//-----------------------------
//Beladestand 1
//-----------------------------
      CALL  "FC_Beladen"
      ( Stand_Nr       := 1,
        E_Belegt       := "DB_BE_Stand".Stand[1].IN_Belegt,
        E_S_innen      := "DB_BE_Stand".Stand[1].IN_innen,
        E_S_aussen     := "DB_BE_Stand".Stand[1].IN_aussen,
        E_S_verriegelt := "DB_BE_Stand".Stand[1].verriegelt,
        E_Freigabe     := "DB_BE_Stand".Stand[1].IN_Freigabe,
        Auto_Delete    := #AutoDelete,
        ext_Delete     := FALSE,
        Del_All        := #DeleteAll,
        Afg_WT_Nr      := false,
        Del_count      := 5
      );

      A     "DB_BE_Stand".Stand[1].OUT_Sperre_in;
      O     #Anforderung_QF;
      =     "DB_POS".POS[25].notFG_in;

// GO links
      L     "DB_POS".POS[27].next_WT;
      L     0;
      <>I;
      S     "DB_POS".POS[25].notFG_in;

      A     "DB_BE_Stand".Stand[1].OUT_Sperre_FW;
      O     #Sperre_TW;
      O(;
      A     "DI_FW_1".ZST.Oben_li;
      A(;
      A     "DB_BE_Stand".Stand[1].IN_Belegt;
      O     "DB_POS".POS[25].belegt;
      AN    "DB_BE_Stand".Stand[1].IN_aussen;
      );
      O;
      A     "DI_FW_1".ZST.Oben_re;
      A(;
      A     "DB_BE_Stand".Stand[2].IN_Belegt;
      O     "DB_POS".POS[26].belegt;
      AN    "DB_BE_Stand".Stand[2].IN_aussen;
      );
      );
      =     "DB_POS".POS[25].Sperre_FW;

      A     "DB_BE_Stand".Stand[1].OUT_Sperre_out;
      O     #Anforderung_QF;
      =     "DB_POS".POS[25].notFG_out;

//-----------------------------
//Beladestand 2
//-----------------------------
      CALL  "FC_Beladen"
      ( Stand_Nr       := 2,
        E_Belegt       := "DB_BE_Stand".Stand[2].IN_Belegt,
        E_S_innen      := "DB_BE_Stand".Stand[2].IN_innen,
        E_S_aussen     := "DB_BE_Stand".Stand[2].IN_aussen,
        E_S_verriegelt := "DB_BE_Stand".Stand[2].verriegelt,
        E_Freigabe     := "DB_BE_Stand".Stand[2].IN_Freigabe,
        Auto_Delete    := #AutoDelete,
        ext_Delete     := FALSE,
        Del_All        := #DeleteAll,
        Afg_WT_Nr      := false,
        Del_count      := 5
      );

      A     "DB_BE_Stand".Stand[2].OUT_Sperre_in;
      O     #Anforderung_QF;
      =     "DB_POS".POS[26].notFG_in;
// GO rechts
      L     "DB_POS".POS[28].next_WT;
      L     0;
      <>I;
      S     "DB_POS".POS[26].notFG_in;

      A     "DB_BE_Stand".Stand[2].OUT_Sperre_out;
      O     #Anforderung_QF;
      =     "DB_POS".POS[26].notFG_out;

//-----------------------------
//Beladestand 3 (GO links)
//-----------------------------
      CALL  "FC_Beladen"
      ( Stand_Nr       := 3,
        E_Belegt       := "DB_BE_Stand".Stand[3].IN_Belegt,
        E_S_innen      := "DB_BE_Stand".Stand[3].IN_innen,
        E_S_aussen     := "DB_BE_Stand".Stand[3].IN_aussen,
        E_S_verriegelt := "DB_BE_Stand".Stand[3].verriegelt,
        E_Freigabe     := "DB_BE_Stand".Stand[3].IN_Freigabe,
        Auto_Delete    := #AutoDelete,
        ext_Delete     := FALSE,
        Del_All        := #DeleteAll,
        Afg_WT_Nr      := false,
        Del_count      := 5
      );

      A     "DB_BE_Stand".Stand[3].OUT_Sperre_in;
      O     #Anforderung_QF;
      =     "DB_POS".POS[27].notFG_in;

//KS links
      L     "DB_POS".POS[25].next_WT;
      L     0;
      <>I;
      O(;
      L     "DB_POS".POS[29].next_WT;
      <>I;
      );
      O(;
      A     "DB_BE_Stand".Stand[1].IN_Belegt;
      A     "DB_BE_Stand".Stand[1].IN_innen;
      );
      O(;
      A     "DB_BE_Stand".Stand[5].IN_Belegt;
      A     "DB_BE_Stand".Stand[5].IN_innen;
      );
      S     "DB_POS".POS[27].notFG_in;

      A     "DB_BE_Stand".Stand[3].OUT_Sperre_out;
      O     #Anforderung_QF;
      =     "DB_POS".POS[27].notFG_out;

//-----------------------------
//Beladestand 4 (GO rechts)
//-----------------------------
      CALL  "FC_Beladen"
      ( Stand_Nr       := 4,
        E_Belegt       := "DB_BE_Stand".Stand[4].IN_Belegt,
        E_S_innen      := "DB_BE_Stand".Stand[4].IN_innen,
        E_S_aussen     := "DB_BE_Stand".Stand[4].IN_aussen,
        E_S_verriegelt := "DB_BE_Stand".Stand[4].verriegelt,
        E_Freigabe     := "DB_BE_Stand".Stand[4].IN_Freigabe,
        Auto_Delete    := #AutoDelete,
        ext_Delete     := FALSE,
        Del_All        := #DeleteAll,
        Afg_WT_Nr      := false,
        Del_count      := 5
      );

      A     "DB_BE_Stand".Stand[4].OUT_Sperre_in;
      O     #Anforderung_QF;
      =     "DB_POS".POS[28].notFG_in;
//KS rechts
      L     "DB_POS".POS[26].next_WT;
      L     0;
      <>I;
      O(;
      L     "DB_POS".POS[30].next_WT;
      <>I;
      );
      O(;
      A     "DB_BE_Stand".Stand[2].IN_Belegt;
      A     "DB_BE_Stand".Stand[2].IN_innen;
      );
      O(;
      A     "DB_BE_Stand".Stand[6].IN_Belegt;
      A     "DB_BE_Stand".Stand[6].IN_innen;
      );
      S     "DB_POS".POS[28].notFG_in;

      A     "DB_BE_Stand".Stand[4].OUT_Sperre_out;
      O     #Anforderung_QF;
      =     "DB_POS".POS[28].notFG_out;

//-------------------------------
//Beladestand 5 (KS hinten links)
//-------------------------------
      CALL  "FC_Beladen"
      ( Stand_Nr       := 5,
        E_Belegt       := "DB_BE_Stand".Stand[5].IN_Belegt,
        E_S_innen      := "DB_BE_Stand".Stand[5].IN_innen,
        E_S_aussen     := "DB_BE_Stand".Stand[5].IN_aussen,
        E_S_verriegelt := "DB_BE_Stand".Stand[5].verriegelt,
        E_Freigabe     := "DB_BE_Stand".Stand[5].IN_Freigabe,
        Auto_Delete    := #AutoDelete,
        ext_Delete     := FALSE,
        Del_All        := #DeleteAll,
        Afg_WT_Nr      := false,
        Del_count      := 5
      );

      L     "DB_POS".POS[25].next_WT;
      L     0;
      <>I;
      O     "DB_BE_Stand".Stand[1].IN_Belegt;
      AN    "DB_BE_Stand".Stand[1].IN_aussen;
      O     "DB_BE_Stand".Stand[5].OUT_Sperre_in;
      O     #Anforderung_QF;
      =     "DB_POS".POS[29].notFG_in;
// GO links
      L     "DB_POS".POS[27].next_WT;
      L     0;
      <>I;
      S     "DB_POS".POS[29].notFG_in;

      A     "DB_BE_Stand".Stand[5].OUT_Sperre_FW;
      O(;
      A     "DB_POS".POS[29].FW_in_POS;
      A(;
      A     "DI_FW_1".ZST.Oben_li;
      A(;
      A     "DB_BE_Stand".Stand[1].IN_Belegt;
      O     "DB_POS".POS[25].belegt;
      AN    "DB_BE_Stand".Stand[1].IN_aussen;
      );
      O;
      A     "DI_FW_1".ZST.Oben_re;
      A(;
      A     "DB_BE_Stand".Stand[2].IN_Belegt;
      O     "DB_POS".POS[26].belegt;
      AN    "DB_BE_Stand".Stand[2].IN_aussen;
      );
      );
      );
      O     #Sperre_TW;
      =     "DB_POS".POS[29].Sperre_FW;

      L     "DB_POS".POS[25].next_WT;
      L     0;
      <>I;
      O     "DB_BE_Stand".Stand[1].IN_Belegt;
      AN    "DB_BE_Stand".Stand[1].IN_aussen;
      O     "DB_BE_Stand".Stand[5].OUT_Sperre_out;
      O     #Anforderung_QF;
      =     "DB_POS".POS[29].notFG_out;

//--------------------------------
//Beladestand 6 (KS hinten rechts)
//--------------------------------
      CALL  "FC_Beladen"
      ( Stand_Nr       := 6,
        E_Belegt       := "DB_BE_Stand".Stand[6].IN_Belegt,
        E_S_innen      := "DB_BE_Stand".Stand[6].IN_innen,
        E_S_aussen     := "DB_BE_Stand".Stand[6].IN_aussen,
        E_S_verriegelt := "DB_BE_Stand".Stand[6].verriegelt,
        E_Freigabe     := "DB_BE_Stand".Stand[6].IN_Freigabe,
        Auto_Delete    := #AutoDelete,
        ext_Delete     := FALSE,
        Del_All        := #DeleteAll,
        Afg_WT_Nr      := false,
        Del_count      := 5
      );


      L     "DB_POS".POS[26].next_WT;
      L     0;
      <>I;
      O     "DB_BE_Stand".Stand[2].IN_Belegt;
      AN    "DB_BE_Stand".Stand[2].IN_aussen;
      O     "DB_BE_Stand".Stand[6].OUT_Sperre_in;
      O     #Anforderung_QF;
      =     "DB_POS".POS[30].notFG_in;
// GO rechts
      L     "DB_POS".POS[28].next_WT;
      L     0;
      <>I;
      S     "DB_POS".POS[30].notFG_in;

      L     "DB_POS".POS[26].next_WT;
      L     0;
      <>I;
      O     "DB_BE_Stand".Stand[2].IN_Belegt;
      AN    "DB_BE_Stand".Stand[2].IN_aussen;
      O     "DB_BE_Stand".Stand[6].OUT_Sperre_out;
      O     #Anforderung_QF;
      =     "DB_POS".POS[30].notFG_out;

END_FUNCTION

FUNCTION "FC_Rez_to_DB45" : Void   // FC1, LAD
TITLE = Füllt nach Aufgabetaste (Panel) Technologie DB
{ S7_Optimized_Access := 'TRUE' }
// stored: SetENOAutomatically true
   VAR_TEMP
      Ptr_Befehl_dyn : Int;
      Ptr_Param_dyn : Int;
      i : Int;
   END_VAR
   VAR CONSTANT
      KS : USInt := 1;   // kurz schmal
      LS : USInt := 2;   // lang schmal
      GO : USInt := 3;   // Großoptik
      Typ_KS : Byte := 16#11;
      Typ_LS : Byte := 16#12;
      Typ_GO : Byte := 16#20;
      Startpos_CM01 : Byte := 16#1;
      Startpos_CM02 : Byte := 16#D;
      Startpos_CM03 : Byte := 16#7;
      Startpos_CM04 : Byte := 16#13;
      Startpos_BE : Byte := 16#19;
      Laenge : Byte := 16#6;
      leer : Byte;
      M_area : Byte := 16#83;
      DB_area : Byte := 16#84;
      Ptr_Befehl_1 : Int := 260;   // Adresse Befehlsparameter
      Ptr_Befehl_2 : Int := 264;   // Adresse Befehlsparameter
      Ptr_Befehl_3 : Int := 268;   // Adresse Befehlsparameter
      Ptr_Befehl_4 : Int := 272;   // Adresse Befehlsparameter
      Ptr_Befehl_5 : Int := 276;   // Adresse Befehlsparameter
      Ptr_Befehl_6 : Int := 280;   // Adresse Befehlsparameter
      Ptr_Befehl_7 : Int;   // Adresse Befehlsparameter
      Techno_DB : DInt := 45;
   END_VAR
BEGIN

REGION Network 1 (SCL): aktuelle Auswahl in Arbeitsstruktur kopieren
   IF "DB_Prog_edit".akt_Aufgabe_Prog <> "DB_Prog_edit".old_Aufgabe_Prog THEN
       "DB_Prog_edit".Prog_Aufgabe.Prog := "DB_Prog_edit".Prog["DB_Prog_edit".akt_Aufgabe_Prog];

       "DB_Prog_edit".old_Aufgabe_Prog := "DB_Prog_edit".akt_Aufgabe_Prog;
   END_IF;
END_REGION

REGION Network 2 (SCL): Artikeldaten für aufgabe aufbereiten
   IF "Panel".Aufgabe.Freigabe AND "DB_Prog_edit".StandNr <> 0  AND "DB_Prog_edit".akt_Aufgabe_Prog <>0  AND "DB_Prog_edit".Prog_Aufgabe.Korb_Nr <>0 THEN

       "DB_Prog_edit".GZ_Charge := "DB_Prog_edit".GZ_Charge + 1; // Gesamtzähler erhöhen
       "DB_Techno".WT_NR_lng := "DB_Prog_edit".GZ_Charge; // Chargenzähler
       "DB_Techno".STAND_NR := "DB_Prog_edit".StandNr; // Nummer B/E-Stand: 1..6
       "DB_Techno".Korb_Nr := INT_TO_USINT("DB_Prog_edit".Prog_Aufgabe.Korb_Nr); // Korb 1..13

       // Modus auswerten
       IF NOT "DB_ANLAGE".config.NormalB THEN
           // Kombi-Mode
           CASE "DB_Prog_edit".Prog_Aufgabe.Korb_Nr OF
               1..3:  // "151" Korb kurz 1..3
                   "DB_Prog_edit".Prog_Aufgabe.Prog.ParaByte.%X4 := TRUE;
                   "DB_Prog_edit".Prog_Aufgabe.Prog.ParaByte.%X5 := FALSE;

               4..8:   // "161" Korb kurz 4..8
                   "DB_Prog_edit".Prog_Aufgabe.Prog.ParaByte.%X4 := FALSE;
                   "DB_Prog_edit".Prog_Aufgabe.Prog.ParaByte.%X5 := TRUE;

               9..11:  // "151" Korb lang 1..3
                   "DB_Prog_edit".Prog_Aufgabe.Prog.ParaByte.%X4 := TRUE;
                   "DB_Prog_edit".Prog_Aufgabe.Prog.ParaByte.%X5 := FALSE;

               12..13:   // "161" Korb lang 4, Großoptik 
                   "DB_Prog_edit".Prog_Aufgabe.Prog.ParaByte.%X4 := FALSE;
                   "DB_Prog_edit".Prog_Aufgabe.Prog.ParaByte.%X5 := TRUE;
           END_CASE;

       ELSE
           // Normalbetrieb
           "DB_Prog_edit".Prog_Aufgabe.Prog.ParaByte.%X4 := FALSE;
           "DB_Prog_edit".Prog_Aufgabe.Prog.ParaByte.%X5 := FALSE;
       END_IF;

       "DB_Techno".Technologie := "DB_Prog_edit".akt_Aufgabe_Prog; // aktuelles Programm: 1..99
           // WT-Typ
       CASE "DB_Prog_edit".Prog_Aufgabe.Prog.Geometrie OF
           #KS:  
               "DB_Techno".WT_Typ := #Typ_KS;
           #LS:  
               "DB_Techno".WT_Typ := #Typ_LS;
           #GO:
               "DB_Techno".WT_Typ := #Typ_GO;
           ELSE
               "DB_Techno".WT_Typ := 0;
       END_CASE;
    // Langsam senken /Langsam heben / Modi
       "DB_Techno".ParaByte := "DB_Prog_edit".Prog_Aufgabe.Prog.ParaByte;

       "DB_Techno".KorrATZ := "DB_Prog_edit".Prog_Aufgabe.Prog.Faktor_ATZ;
       "DB_Techno".KorrPend := 1.0;


       // Normal-Betrieb - nur Ware "151" Gruppe CM01/CM02
       IF "DB_ANLAGE".config.NormalB THEN
           REGION NormalB
               // Vorspülen
               #Ptr_Befehl_dyn := 1;
               #Ptr_Param_dyn := 340;

               "DB_Techno".stBefehle[#Ptr_Befehl_dyn].Kennung := #Startpos_CM03;
               "DB_Techno".stBefehle[#Ptr_Befehl_dyn].FirstPos1 := #Startpos_CM03;
               "DB_Techno".stBefehle[#Ptr_Befehl_dyn].Grpleng1 := #Laenge;
               "DB_Techno".stBefehle[#Ptr_Befehl_dyn].FirstPos2 := #leer;
               "DB_Techno".stBefehle[#Ptr_Befehl_dyn].Grpleng2 := #leer;
               "DB_Techno".stBefehle[#Ptr_Befehl_dyn].Merker := #leer;
               "DB_Techno".stBefehle[#Ptr_Befehl_dyn].Param_Ptr := #Ptr_Param_dyn; //#Ptr_Befehl_1;
               "temp_Sollzeit" := TOD_TO_DINT("DB_Prog_edit".Prog_Aufgabe.Prog.CM03_VorSpuel.Expo) / 1000;

               POKE_BLK(area_src := #M_area,
                        dbNumber_src := 0,
                        byteOffset_src := 256,
                        area_dest := #DB_area,
                        dbNumber_dest := #Techno_DB,
                        byteOffset_dest := #Ptr_Param_dyn, //Ptr_Befehl_1,
                        count := 4);

               // Vorätzen
               IF "DB_Prog_edit".Prog_Aufgabe.Prog.CM01_VorAetz.Anzahl_Voraetz > 0 THEN
                   FOR #i := 1 TO BYTE_TO_INT("DB_Prog_edit".Prog_Aufgabe.Prog.CM01_VorAetz.Anzahl_Voraetz) DO
                       #Ptr_Befehl_dyn := #Ptr_Befehl_dyn + 1;
                       #Ptr_Param_dyn := #Ptr_Param_dyn + 4;

                       "DB_Techno".stBefehle[#Ptr_Befehl_dyn].Kennung := #Startpos_CM01;
                       "DB_Techno".stBefehle[#Ptr_Befehl_dyn].FirstPos1 := #Startpos_CM01;
                       "DB_Techno".stBefehle[#Ptr_Befehl_dyn].Grpleng1 := #Laenge;
                       "DB_Techno".stBefehle[#Ptr_Befehl_dyn].FirstPos2 := #Startpos_CM02;
                       "DB_Techno".stBefehle[#Ptr_Befehl_dyn].Grpleng2 := #Laenge;
                       "DB_Techno".stBefehle[#Ptr_Befehl_dyn].Merker := #leer;
                       "DB_Techno".stBefehle[#Ptr_Befehl_dyn].Param_Ptr := #Ptr_Param_dyn; // #Ptr_Befehl_2;
                       "temp_Sollzeit" := TOD_TO_DINT("DB_Prog_edit".Prog_Aufgabe.Prog.CM01_VorAetz.Expo) / 1000;

                       POKE_BLK(area_src := #M_area,
                                dbNumber_src := 0,
                                byteOffset_src := 256,
                                area_dest := #DB_area,
                                dbNumber_dest := #Techno_DB,
                                byteOffset_dest := #Ptr_Param_dyn, //Ptr_Befehl_2,
                                count := 4);


                       // Spülen Vorätzen
                       #Ptr_Befehl_dyn := #Ptr_Befehl_dyn + 1;
                       #Ptr_Param_dyn := #Ptr_Param_dyn + 4;

                       "DB_Techno".stBefehle[#Ptr_Befehl_dyn].Kennung := #Startpos_CM03;
                       "DB_Techno".stBefehle[#Ptr_Befehl_dyn].FirstPos1 := #Startpos_CM03;
                       "DB_Techno".stBefehle[#Ptr_Befehl_dyn].Grpleng1 := #Laenge;
                       "DB_Techno".stBefehle[#Ptr_Befehl_dyn].FirstPos2 := #leer;
                       "DB_Techno".stBefehle[#Ptr_Befehl_dyn].Grpleng2 := #leer;
                       "DB_Techno".stBefehle[#Ptr_Befehl_dyn].Merker := #leer;
                       "DB_Techno".stBefehle[#Ptr_Befehl_dyn].Param_Ptr := #Ptr_Param_dyn; // #Ptr_Befehl_3;
                       "temp_Sollzeit" := TOD_TO_DINT("DB_Prog_edit".Prog_Aufgabe.Prog.CM03_SpuelVorAetz.Expo) / 1000;

                       POKE_BLK(area_src := #M_area,
                                dbNumber_src := 0,
                                byteOffset_src := 256,
                                area_dest := #DB_area,
                                dbNumber_dest := #Techno_DB,
                                byteOffset_dest := #Ptr_Param_dyn, //#Ptr_Befehl_3,
                                count := 4);

                   END_FOR;
               END_IF;

               // Ätzen
               #Ptr_Befehl_dyn := #Ptr_Befehl_dyn + 1;
               #Ptr_Param_dyn := #Ptr_Param_dyn + 4;

               "DB_Techno".stBefehle[#Ptr_Befehl_dyn].Kennung := #Startpos_CM01;
               "DB_Techno".stBefehle[#Ptr_Befehl_dyn].FirstPos1 := #Startpos_CM01;
               "DB_Techno".stBefehle[#Ptr_Befehl_dyn].Grpleng1 := #Laenge;
               "DB_Techno".stBefehle[#Ptr_Befehl_dyn].FirstPos2 := #Startpos_CM02;
               "DB_Techno".stBefehle[#Ptr_Befehl_dyn].Grpleng2 := #Laenge;
               "DB_Techno".stBefehle[#Ptr_Befehl_dyn].Merker := #leer;
               "DB_Techno".stBefehle[#Ptr_Befehl_dyn].Param_Ptr := #Ptr_Param_dyn; //#Ptr_Befehl_4;
               "temp_Sollzeit" := TOD_TO_DINT("DB_Prog_edit".Prog_Aufgabe.Prog.CM01_Aetzen.Expo) / 1000;

               POKE_BLK(area_src := #M_area,
                        dbNumber_src := 0,
                        byteOffset_src := 256,
                        area_dest := #DB_area,
                        dbNumber_dest := #Techno_DB,
                        byteOffset_dest := #Ptr_Param_dyn, //#Ptr_Befehl_4,
                        count := 4);

               // Spülen 1 Ätzen
               #Ptr_Befehl_dyn := #Ptr_Befehl_dyn + 1;
               #Ptr_Param_dyn := #Ptr_Param_dyn + 4;

               "DB_Techno".stBefehle[#Ptr_Befehl_dyn].Kennung := #Startpos_CM03;
               "DB_Techno".stBefehle[#Ptr_Befehl_dyn].FirstPos1 := #Startpos_CM03;
               "DB_Techno".stBefehle[#Ptr_Befehl_dyn].Grpleng1 := #Laenge;
               "DB_Techno".stBefehle[#Ptr_Befehl_dyn].FirstPos2 := #leer;
               "DB_Techno".stBefehle[#Ptr_Befehl_dyn].Grpleng2 := #leer;
               "DB_Techno".stBefehle[#Ptr_Befehl_dyn].Merker := #leer;
               "DB_Techno".stBefehle[#Ptr_Befehl_dyn].Param_Ptr := #Ptr_Param_dyn; //#Ptr_Befehl_5;
               "temp_Sollzeit" := TOD_TO_DINT("DB_Prog_edit".Prog_Aufgabe.Prog.CM03_Spl_1.Expo) / 1000;

               POKE_BLK(area_src := #M_area,
                        dbNumber_src := 0,
                        byteOffset_src := 256,
                        area_dest := #DB_area,
                        dbNumber_dest := #Techno_DB,
                        byteOffset_dest := #Ptr_Param_dyn, //#Ptr_Befehl_5,
                        count := 4);

               // Spülen 2 Ätzen
               #Ptr_Befehl_dyn := #Ptr_Befehl_dyn + 1;
               #Ptr_Param_dyn := #Ptr_Param_dyn + 4;

               "DB_Techno".stBefehle[#Ptr_Befehl_dyn].Kennung := #Startpos_CM04;
               "DB_Techno".stBefehle[#Ptr_Befehl_dyn].FirstPos1 := #Startpos_CM04;
               "DB_Techno".stBefehle[#Ptr_Befehl_dyn].Grpleng1 := #Laenge;
               "DB_Techno".stBefehle[#Ptr_Befehl_dyn].FirstPos2 := #leer;
               "DB_Techno".stBefehle[#Ptr_Befehl_dyn].Grpleng2 := #leer;
               "DB_Techno".stBefehle[#Ptr_Befehl_dyn].Merker := #leer;
               "DB_Techno".stBefehle[#Ptr_Befehl_dyn].Param_Ptr := #Ptr_Param_dyn; //#Ptr_Befehl_6;
               "temp_Sollzeit" := TOD_TO_DINT("DB_Prog_edit".Prog_Aufgabe.Prog.CM04_Spl_2.Expo) / 1000;

               POKE_BLK(area_src := #M_area,
                        dbNumber_src := 0,
                        byteOffset_src := 256,
                        area_dest := #DB_area,
                        dbNumber_dest := #Techno_DB,
                        byteOffset_dest := #Ptr_Param_dyn, //#Ptr_Befehl_6,
                        count := 4);
           END_REGION

       ELSE // Kombi-Modus: "151" CM02 / CM04 ; "161" CM01 / CM03


           IF  "DB_Prog_edit".Prog_Aufgabe.Prog.ParaByte.%X4 THEN
            REGION WT_151                    
                // Vorspülen             
                  #Ptr_Befehl_dyn := 1;
                  #Ptr_Param_dyn := 340;

                  "DB_Techno".stBefehle[#Ptr_Befehl_dyn].Kennung := #Startpos_CM04;
                   "DB_Techno".stBefehle[#Ptr_Befehl_dyn].FirstPos1 := #Startpos_CM04;
                   "DB_Techno".stBefehle[#Ptr_Befehl_dyn].Grpleng1 := #Laenge;
                   "DB_Techno".stBefehle[#Ptr_Befehl_dyn].FirstPos2 := #leer;
                   "DB_Techno".stBefehle[#Ptr_Befehl_dyn].Grpleng2 := #leer;
                   "DB_Techno".stBefehle[#Ptr_Befehl_dyn].Merker := #leer;
                   "DB_Techno".stBefehle[#Ptr_Befehl_dyn].Param_Ptr := #Ptr_Param_dyn; //#Ptr_Befehl_1;
                   "temp_Sollzeit" := TOD_TO_DINT("DB_Prog_edit".Prog_Aufgabe.Prog.CM03_VorSpuel.Expo) / 1000;

                   POKE_BLK(area_src := #M_area,
                            dbNumber_src := 0,
                            byteOffset_src := 256,
                            area_dest := #DB_area,
                            dbNumber_dest := #Techno_DB,
                            byteOffset_dest := #Ptr_Param_dyn, //Ptr_Befehl_1,
                            count := 4);

                   // Vorätzen
                   IF "DB_Prog_edit".Prog_Aufgabe.Prog.CM01_VorAetz.Anzahl_Voraetz > 0 THEN
                       FOR #i := 1 TO BYTE_TO_INT("DB_Prog_edit".Prog_Aufgabe.Prog.CM01_VorAetz.Anzahl_Voraetz) DO
                           #Ptr_Befehl_dyn := #Ptr_Befehl_dyn + 1;
                           #Ptr_Param_dyn := #Ptr_Param_dyn + 4;

                           "DB_Techno".stBefehle[#Ptr_Befehl_dyn].Kennung := #Startpos_CM02;
                           "DB_Techno".stBefehle[#Ptr_Befehl_dyn].FirstPos1 := #Startpos_CM02;
                           "DB_Techno".stBefehle[#Ptr_Befehl_dyn].Grpleng1 := #Laenge;
                           "DB_Techno".stBefehle[#Ptr_Befehl_dyn].FirstPos2 := #leer;
                           "DB_Techno".stBefehle[#Ptr_Befehl_dyn].Grpleng2 := #leer;
                           "DB_Techno".stBefehle[#Ptr_Befehl_dyn].Merker := #leer;
                           "DB_Techno".stBefehle[#Ptr_Befehl_dyn].Param_Ptr := #Ptr_Param_dyn; // #Ptr_Befehl_2;
                           "temp_Sollzeit" := TOD_TO_DINT("DB_Prog_edit".Prog_Aufgabe.Prog.CM01_VorAetz.Expo) / 1000;

                           POKE_BLK(area_src := #M_area,
                                    dbNumber_src := 0,
                                    byteOffset_src := 256,
                                    area_dest := #DB_area,
                                    dbNumber_dest := #Techno_DB,
                                    byteOffset_dest := #Ptr_Param_dyn, //Ptr_Befehl_2,
                                    count := 4);

                           // Spülen Vorätzen
                           #Ptr_Befehl_dyn := #Ptr_Befehl_dyn + 1;
                           #Ptr_Param_dyn := #Ptr_Param_dyn + 4;

                           "DB_Techno".stBefehle[#Ptr_Befehl_dyn].Kennung := #Startpos_CM04;
                           "DB_Techno".stBefehle[#Ptr_Befehl_dyn].FirstPos1 := #Startpos_CM04;
                           "DB_Techno".stBefehle[#Ptr_Befehl_dyn].Grpleng1 := #Laenge;
                           "DB_Techno".stBefehle[#Ptr_Befehl_dyn].FirstPos2 := #leer;
                           "DB_Techno".stBefehle[#Ptr_Befehl_dyn].Grpleng2 := #leer;
                           "DB_Techno".stBefehle[#Ptr_Befehl_dyn].Merker := #leer;
                           "DB_Techno".stBefehle[#Ptr_Befehl_dyn].Param_Ptr := #Ptr_Param_dyn; // #Ptr_Befehl_3;
                           "temp_Sollzeit" := TOD_TO_DINT("DB_Prog_edit".Prog_Aufgabe.Prog.CM03_SpuelVorAetz.Expo) / 1000;

                           POKE_BLK(area_src := #M_area,
                                    dbNumber_src := 0,
                                    byteOffset_src := 256,
                                    area_dest := #DB_area,
                                    dbNumber_dest := #Techno_DB,
                                    byteOffset_dest := #Ptr_Param_dyn, //#Ptr_Befehl_3,
                                    count := 4);

                       END_FOR;
                   END_IF;

                   // Ätzen
                   #Ptr_Befehl_dyn := #Ptr_Befehl_dyn + 1;
                   #Ptr_Param_dyn := #Ptr_Param_dyn + 4;

                   "DB_Techno".stBefehle[#Ptr_Befehl_dyn].Kennung := #Startpos_CM02;
                   "DB_Techno".stBefehle[#Ptr_Befehl_dyn].FirstPos1 := #Startpos_CM02;
                   "DB_Techno".stBefehle[#Ptr_Befehl_dyn].Grpleng1 := #Laenge;
                   "DB_Techno".stBefehle[#Ptr_Befehl_dyn].FirstPos2 := #leer;
                   "DB_Techno".stBefehle[#Ptr_Befehl_dyn].Grpleng2 := #leer;
                   "DB_Techno".stBefehle[#Ptr_Befehl_dyn].Merker := #leer;
                   "DB_Techno".stBefehle[#Ptr_Befehl_dyn].Param_Ptr := #Ptr_Param_dyn; //#Ptr_Befehl_4;
                   "temp_Sollzeit" := TOD_TO_DINT("DB_Prog_edit".Prog_Aufgabe.Prog.CM01_Aetzen.Expo) / 1000;

                   POKE_BLK(area_src := #M_area,
                            dbNumber_src := 0,
                            byteOffset_src := 256,
                            area_dest := #DB_area,
                            dbNumber_dest := #Techno_DB,
                            byteOffset_dest := #Ptr_Param_dyn, //#Ptr_Befehl_4,
                            count := 4);

                   // Spülen 1 Ätzen
                   #Ptr_Befehl_dyn := #Ptr_Befehl_dyn + 1;
                   #Ptr_Param_dyn := #Ptr_Param_dyn + 4;

                   "DB_Techno".stBefehle[#Ptr_Befehl_dyn].Kennung := #Startpos_CM04;
                   "DB_Techno".stBefehle[#Ptr_Befehl_dyn].FirstPos1 := #Startpos_CM04;
                   "DB_Techno".stBefehle[#Ptr_Befehl_dyn].Grpleng1 := #Laenge;
                   "DB_Techno".stBefehle[#Ptr_Befehl_dyn].FirstPos2 := #leer;
                   "DB_Techno".stBefehle[#Ptr_Befehl_dyn].Grpleng2 := #leer;
                   "DB_Techno".stBefehle[#Ptr_Befehl_dyn].Merker := #leer;
                   "DB_Techno".stBefehle[#Ptr_Befehl_dyn].Param_Ptr := #Ptr_Param_dyn; //#Ptr_Befehl_5;
                   "temp_Sollzeit" := TOD_TO_DINT("DB_Prog_edit".Prog_Aufgabe.Prog.CM03_Spl_1.Expo) / 1000;

                   POKE_BLK(area_src := #M_area,
                            dbNumber_src := 0,
                            byteOffset_src := 256,
                            area_dest := #DB_area,
                            dbNumber_dest := #Techno_DB,
                            byteOffset_dest := #Ptr_Param_dyn, //#Ptr_Befehl_5,
                            count := 4);

                   // Spülen 2 Ätzen
                   #Ptr_Befehl_dyn := #Ptr_Befehl_dyn + 1;
                   #Ptr_Param_dyn := #Ptr_Param_dyn + 4;

                   "DB_Techno".stBefehle[#Ptr_Befehl_dyn].Kennung := #Startpos_CM04;
                   "DB_Techno".stBefehle[#Ptr_Befehl_dyn].FirstPos1 := #Startpos_CM04;
                   "DB_Techno".stBefehle[#Ptr_Befehl_dyn].Grpleng1 := #Laenge;
                   "DB_Techno".stBefehle[#Ptr_Befehl_dyn].FirstPos2 := #leer;
                   "DB_Techno".stBefehle[#Ptr_Befehl_dyn].Grpleng2 := #leer;
                   "DB_Techno".stBefehle[#Ptr_Befehl_dyn].Merker := #leer;
                   "DB_Techno".stBefehle[#Ptr_Befehl_dyn].Param_Ptr := #Ptr_Param_dyn; //#Ptr_Befehl_6;
                   "temp_Sollzeit" := TOD_TO_DINT("DB_Prog_edit".Prog_Aufgabe.Prog.CM04_Spl_2.Expo) / 1000;

                   POKE_BLK(area_src := #M_area,
                            dbNumber_src := 0,
                            byteOffset_src := 256,
                            area_dest := #DB_area,
                            dbNumber_dest := #Techno_DB,
                            byteOffset_dest := #Ptr_Param_dyn, //#Ptr_Befehl_6,
                            count := 4);
               END_REGION

           ELSE
            REGION WT_161                    
                   // Vorspülen             
                   #Ptr_Befehl_dyn := 1;
                   #Ptr_Param_dyn := 340;

                   "DB_Techno".stBefehle[#Ptr_Befehl_dyn].Kennung := #Startpos_CM03;
                   "DB_Techno".stBefehle[#Ptr_Befehl_dyn].FirstPos1 := #Startpos_CM03;
                   "DB_Techno".stBefehle[#Ptr_Befehl_dyn].Grpleng1 := #Laenge;
                   "DB_Techno".stBefehle[#Ptr_Befehl_dyn].FirstPos2 := #leer;
                   "DB_Techno".stBefehle[#Ptr_Befehl_dyn].Grpleng2 := #leer;
                   "DB_Techno".stBefehle[#Ptr_Befehl_dyn].Merker := #leer;
                   "DB_Techno".stBefehle[#Ptr_Befehl_dyn].Param_Ptr := #Ptr_Param_dyn; //#Ptr_Befehl_1;
                   "temp_Sollzeit" := TOD_TO_DINT("DB_Prog_edit".Prog_Aufgabe.Prog.CM03_VorSpuel.Expo) / 1000;

                   POKE_BLK(area_src := #M_area,
                            dbNumber_src := 0,
                            byteOffset_src := 256,
                            area_dest := #DB_area,
                            dbNumber_dest := #Techno_DB,
                            byteOffset_dest := #Ptr_Param_dyn, //Ptr_Befehl_1,
                            count := 4);

                   // Vorätzen
                   IF "DB_Prog_edit".Prog_Aufgabe.Prog.CM01_VorAetz.Anzahl_Voraetz > 0 THEN
                       FOR #i := 1 TO BYTE_TO_INT("DB_Prog_edit".Prog_Aufgabe.Prog.CM01_VorAetz.Anzahl_Voraetz) DO
                           #Ptr_Befehl_dyn := #Ptr_Befehl_dyn + 1;
                           #Ptr_Param_dyn := #Ptr_Param_dyn + 4;

                           "DB_Techno".stBefehle[#Ptr_Befehl_dyn].Kennung := #Startpos_CM01;
                           "DB_Techno".stBefehle[#Ptr_Befehl_dyn].FirstPos1 := #Startpos_CM01;
                           "DB_Techno".stBefehle[#Ptr_Befehl_dyn].Grpleng1 := #Laenge;
                           "DB_Techno".stBefehle[#Ptr_Befehl_dyn].FirstPos2 := #leer;
                           "DB_Techno".stBefehle[#Ptr_Befehl_dyn].Grpleng2 := #leer;
                           "DB_Techno".stBefehle[#Ptr_Befehl_dyn].Merker := #leer;
                           "DB_Techno".stBefehle[#Ptr_Befehl_dyn].Param_Ptr := #Ptr_Param_dyn; // #Ptr_Befehl_2;
                           "temp_Sollzeit" := TOD_TO_DINT("DB_Prog_edit".Prog_Aufgabe.Prog.CM01_VorAetz.Expo) / 1000;

                           POKE_BLK(area_src := #M_area,
                                    dbNumber_src := 0,
                                    byteOffset_src := 256,
                                    area_dest := #DB_area,
                                    dbNumber_dest := #Techno_DB,
                                    byteOffset_dest := #Ptr_Param_dyn, //Ptr_Befehl_2,
                                    count := 4);

                           // Spülen Vorätzen
                           #Ptr_Befehl_dyn := #Ptr_Befehl_dyn + 1;
                           #Ptr_Param_dyn := #Ptr_Param_dyn + 4;

                           "DB_Techno".stBefehle[#Ptr_Befehl_dyn].Kennung := #Startpos_CM03;
                           "DB_Techno".stBefehle[#Ptr_Befehl_dyn].FirstPos1 := #Startpos_CM03;
                           "DB_Techno".stBefehle[#Ptr_Befehl_dyn].Grpleng1 := #Laenge;
                           "DB_Techno".stBefehle[#Ptr_Befehl_dyn].FirstPos2 := #leer;
                           "DB_Techno".stBefehle[#Ptr_Befehl_dyn].Grpleng2 := #leer;
                           "DB_Techno".stBefehle[#Ptr_Befehl_dyn].Merker := #leer;
                           "DB_Techno".stBefehle[#Ptr_Befehl_dyn].Param_Ptr := #Ptr_Param_dyn; // #Ptr_Befehl_3;
                           "temp_Sollzeit" := TOD_TO_DINT("DB_Prog_edit".Prog_Aufgabe.Prog.CM03_SpuelVorAetz.Expo) / 1000;

                           POKE_BLK(area_src := #M_area,
                                    dbNumber_src := 0,
                                    byteOffset_src := 256,
                                    area_dest := #DB_area,
                                    dbNumber_dest := #Techno_DB,
                                    byteOffset_dest := #Ptr_Param_dyn, //#Ptr_Befehl_3,
                                    count := 4);

                       END_FOR;
                   END_IF;

                   // Ätzen
                   #Ptr_Befehl_dyn := #Ptr_Befehl_dyn + 1;
                   #Ptr_Param_dyn := #Ptr_Param_dyn + 4;

                   "DB_Techno".stBefehle[#Ptr_Befehl_dyn].Kennung := #Startpos_CM01;
                   "DB_Techno".stBefehle[#Ptr_Befehl_dyn].FirstPos1 := #Startpos_CM01;
                   "DB_Techno".stBefehle[#Ptr_Befehl_dyn].Grpleng1 := #Laenge;
                   "DB_Techno".stBefehle[#Ptr_Befehl_dyn].FirstPos2 := #leer;
                   "DB_Techno".stBefehle[#Ptr_Befehl_dyn].Grpleng2 := #leer;
                   "DB_Techno".stBefehle[#Ptr_Befehl_dyn].Merker := #leer;
                   "DB_Techno".stBefehle[#Ptr_Befehl_dyn].Param_Ptr := #Ptr_Param_dyn; //#Ptr_Befehl_4;
                   "temp_Sollzeit" := TOD_TO_DINT("DB_Prog_edit".Prog_Aufgabe.Prog.CM01_Aetzen.Expo) / 1000;

                   POKE_BLK(area_src := #M_area,
                            dbNumber_src := 0,
                            byteOffset_src := 256,
                            area_dest := #DB_area,
                            dbNumber_dest := #Techno_DB,
                            byteOffset_dest := #Ptr_Param_dyn, //#Ptr_Befehl_4,
                            count := 4);

                   // Spülen 1 Ätzen
                   #Ptr_Befehl_dyn := #Ptr_Befehl_dyn + 1;
                   #Ptr_Param_dyn := #Ptr_Param_dyn + 4;

                   "DB_Techno".stBefehle[#Ptr_Befehl_dyn].Kennung := #Startpos_CM03;
                   "DB_Techno".stBefehle[#Ptr_Befehl_dyn].FirstPos1 := #Startpos_CM03;
                   "DB_Techno".stBefehle[#Ptr_Befehl_dyn].Grpleng1 := #Laenge;
                   "DB_Techno".stBefehle[#Ptr_Befehl_dyn].FirstPos2 := #leer;
                   "DB_Techno".stBefehle[#Ptr_Befehl_dyn].Grpleng2 := #leer;
                   "DB_Techno".stBefehle[#Ptr_Befehl_dyn].Merker := #leer;
                   "DB_Techno".stBefehle[#Ptr_Befehl_dyn].Param_Ptr := #Ptr_Param_dyn; //#Ptr_Befehl_5;
                   "temp_Sollzeit" := TOD_TO_DINT("DB_Prog_edit".Prog_Aufgabe.Prog.CM03_Spl_1.Expo) / 1000;

                   POKE_BLK(area_src := #M_area,
                            dbNumber_src := 0,
                            byteOffset_src := 256,
                            area_dest := #DB_area,
                            dbNumber_dest := #Techno_DB,
                            byteOffset_dest := #Ptr_Param_dyn, //#Ptr_Befehl_5,
                            count := 4);

                   // Spülen 2 Ätzen
                   #Ptr_Befehl_dyn := #Ptr_Befehl_dyn + 1;
                   #Ptr_Param_dyn := #Ptr_Param_dyn + 4;

                   "DB_Techno".stBefehle[#Ptr_Befehl_dyn].Kennung := #Startpos_CM03;
                   "DB_Techno".stBefehle[#Ptr_Befehl_dyn].FirstPos1 := #Startpos_CM03;
                   "DB_Techno".stBefehle[#Ptr_Befehl_dyn].Grpleng1 := #Laenge;
                   "DB_Techno".stBefehle[#Ptr_Befehl_dyn].FirstPos2 := #leer;
                   "DB_Techno".stBefehle[#Ptr_Befehl_dyn].Grpleng2 := #leer;
                   "DB_Techno".stBefehle[#Ptr_Befehl_dyn].Merker := #leer;
                   "DB_Techno".stBefehle[#Ptr_Befehl_dyn].Param_Ptr := #Ptr_Param_dyn; //#Ptr_Befehl_6;
                   "temp_Sollzeit" := TOD_TO_DINT("DB_Prog_edit".Prog_Aufgabe.Prog.CM04_Spl_2.Expo) / 1000;

                   POKE_BLK(area_src := #M_area,
                            dbNumber_src := 0,
                            byteOffset_src := 256,
                            area_dest := #DB_area,
                            dbNumber_dest := #Techno_DB,
                            byteOffset_dest := #Ptr_Param_dyn, //#Ptr_Befehl_6,
                            count := 4);
               END_REGION

            END_IF;

       END_IF;

       // Ausfahrt
       #Ptr_Befehl_dyn := #Ptr_Befehl_dyn + 1;
       #Ptr_Param_dyn := #Ptr_Param_dyn + 4;

       "DB_Techno".stBefehle[#Ptr_Befehl_dyn].Kennung := #Startpos_BE;
       "DB_Techno".stBefehle[#Ptr_Befehl_dyn].FirstPos1 := #Startpos_BE;
       "DB_Techno".stBefehle[#Ptr_Befehl_dyn].Grpleng1 := #Laenge;
       "DB_Techno".stBefehle[#Ptr_Befehl_dyn].FirstPos2 := #leer;
       "DB_Techno".stBefehle[#Ptr_Befehl_dyn].Grpleng2 := #leer;
       "DB_Techno".stBefehle[#Ptr_Befehl_dyn].Merker := #leer;
       "DB_Techno".stBefehle[#Ptr_Befehl_dyn].Param_Ptr := #Ptr_Param_dyn; //#Ptr_Befehl_7;

       // Ende
       #Ptr_Befehl_dyn := #Ptr_Befehl_dyn + 1;

       FOR #i := #Ptr_Befehl_dyn TO 20 DO
            #Ptr_Befehl_dyn := #i;
            // #Ptr_Param_dyn := #Ptr_Param_dyn + 4;

           "DB_Techno".stBefehle[#Ptr_Befehl_dyn].Kennung := #leer;
           "DB_Techno".stBefehle[#Ptr_Befehl_dyn].FirstPos1 := #leer;
           "DB_Techno".stBefehle[#Ptr_Befehl_dyn].Grpleng1 := #leer;
           "DB_Techno".stBefehle[#Ptr_Befehl_dyn].FirstPos2 := #leer;
           "DB_Techno".stBefehle[#Ptr_Befehl_dyn].Grpleng2 := #leer;
           "DB_Techno".stBefehle[#Ptr_Befehl_dyn].Merker := #leer;
           "DB_Techno".stBefehle[#Ptr_Befehl_dyn].Param_Ptr := 0;
       END_FOR;

       "DB_Techno".Name := "DB_Prog_edit".Prog_Aufgabe.Prog.Name;

       "DB_Techno".DATEN_gueltig := "Panel".Aufgabe.Freigabe;
       // Rücksetzen
       "Panel".Aufgabe.Freigabe := FALSE;
       "DB_Prog_edit".StandNr := 0;
       "DB_Prog_edit".Variante := 0;
       "DB_Prog_edit".Prog_Aufgabe.Korb_Nr := 0;

   END_IF;
END_REGION
END_FUNCTION

FUNCTION "FC_AEND_WT" : Void   // FC45, STL
TITLE = WT-Daten neu/geändert
{ S7_Optimized_Access := 'FALSE' }
AUTHOR : MS
// Laden von WT-Daten aus Übergabepuffer
// stored: AutoNumber false
   VAR_TEMP
      WT_lang : DWord;
      WT_Nr_lang : DWord;
      WT_DB : Int;
      Quell_DB : Int;
      last_WT_DB : Int;
      Beginn_Daten : Int;
      Ende_daten : Int;
      Stand_Nr : USInt;
      Pos_Nr : USInt;
      WT_Nr : Byte;
      WT_kurz : Byte;
      inf_1 : Byte;
      WTnew : Bool;   // Warenträger neu
      "Return" : Bool;
      Stand_ok : Bool;
      WT_nok : Bool;
      neuAufgabe : Bool;
      Del_All : Bool;
   END_VAR
BEGIN

NETWORK
TITLE = Test gibt es neue Daten
// -gibt es neue Daten
// -wo stehen diese
// -handelt es sich um Aktualisierungsdaten
//-------------------------------
//Neue Daten?
//-------------------------------
      A     "DB_Techno".DATEN_gueltig;
      L     S5T#20S;
      SD    "T_Aend_WT";

      A     "DB_Techno".DATEN_gueltig;
      A     "T_Aend_WT";
      R     "DB_Techno".DATEN_gueltig;
//-------------------------------
//keine neuen Daten
//-------------------------------
      AN    "DB_Techno".DATEN_gueltig;
      BEC;
      SET;
      R     #Stand_ok;
      R     #Del_All;

//----------------------------------
//Handelt es sich um eine Neuaufgabe
//----------------------------------
      L     "DB_Techno".STAND_NR;
      T     #Stand_Nr;
      L     0;
      <>I;
      =     #WTnew;
      =     #neuAufgabe;
      JC    New;
      JU    Old;


NETWORK
TITLE = Neuer WT
//------------------------
//Stand-Nr prüfen
//------------------------
New:  L     "DB_BE_Stand".Anzahl;
      L     #Stand_Nr;
      <I;
      JC    ende;

      OPN   "DB_BE_Stand";
      A     "DB_BE_Stand".Stand[#Stand_Nr].Del_All;
      =     #Del_All;
      L     0;
      L     "DB_BE_Stand".Stand[#Stand_Nr].Pos_Nr;
      ==I;
      JC    ende;
      S     #Stand_ok;
//------------------------
//Pos auf WT testen
//------------------------
      T     #Pos_Nr;
      L     0;
      L     "DB_POS".POS[#Pos_Nr].WT_DB;
      ==I;
      JC    WTck;
      T     #WT_Nr;
      L     100;
      +I;
      T     #WT_DB;
      JU    load;
//------------------------
//Neuen WT suchen
//------------------------
WTck: AN    #Del_All;  //keinen neuen WT suchen
      JC    ende;
      L     "DB_ANLAGE".config.ANZ_WT;
      L     100;
      +I;
      T     #last_WT_DB;
      L     101;
      T     #WT_DB;
ret:  OPN   DB [#WT_DB];
      L     %DBB15;
      L     0;
      ==I;
      JC    fnd;
      L     #WT_DB;
      L     1;
      +I;
      T     #WT_DB;
      L     #last_WT_DB;
      >I;
      JC    ende;
      JU    ret;
fnd:  L     #WT_DB;
      L     100;
      -I;
      T     #WT_Nr;
      JU    load;


NETWORK
TITLE = Alter WT
// Aktualisieren
//-------------------------------
//prüfen ob WT_Nr gültig
//-------------------------------
Old:  L     "DB_Techno".WT_NR_kurz;
      T     #WT_Nr;
      L     "DB_ANLAGE".config.ANZ_WT;
      >I;
      JC    ende;
      L     0;
      L     #WT_Nr;
      >=I;
      JC    ende;
      L     100;
      +I;
      T     #WT_DB;
//-------------------------------
//passen die WT-Daten zueinander
//-------------------------------
      L     "DB_Techno".WT_NR_lng;
      OPN   DB [#WT_DB];
      L     %DBD6;  // WT-Nr lang
      <>D;
      JC    ende;
      L     %DBB15;  //"DB_WTx".POS
      T     #Pos_Nr;

load: NOP   0;

NETWORK
TITLE = Daten laden
//------------------------
//allgemeine Daten laden
//------------------------
ldok: L     "DB_Techno".Beginn_Daten;
      T     #Beginn_Daten;
      L     "DB_Techno".Ende_Daten;
      T     #Ende_daten;

      CALL  "FC_DB_COPY"
      ( CLR_ALT_DB := FALSE,
        ALT_DB     := 45,
        NEU_DB     := #WT_DB,
        COPY_START := #Beginn_Daten,
        COPY_ENDE  := #Ende_daten,
        ZIEL_START := 78,  // HCA: Namen mit kopieren
        CLR_START  := 0,
        CLR_ENDE   := 0,
        START      := "DB_Techno".DATEN_gueltig
      );

      L     "DB_Techno".Prioritaet;
      L     0;
      <>I;
      OPN   DB [#WT_DB];
      =     %DBX18.0;  //PRIORITÄT

      OPN   DB [#WT_DB];
      A     %DBX18.1;  //"DB_WT1".in_Anlage
      R     #neuAufgabe;  //WT wurde bereits neu aufgegeben

      A     %DBX22.3;  //"DB_WT1".WT_nok
      AN    #Stand_ok;
      =     #WT_nok;  //nok merken

      L     "DB_Techno".ParaByte;  //Parameterinfo laden
      OPN   DB [#WT_DB];
      T     %DBB22;
      L     "DB_Techno".WT_NR_lng;
      OPN   DB [#WT_DB];
      T     %DBD6;  //WT_Nr_lang
      T     #WT_Nr_lang;
      L     "DB_Techno".Speed_Up;
      OPN   DB [#WT_DB];
      T     %DBW64;  //"DB_WT1".Speed_Up
      L     "DB_Techno".Speed_Dn;
      OPN   DB [#WT_DB];
      T     %DBW66;  //"DB_WT1".Speed_Dn
      L     "DB_Techno".Speed_Fahrt;
      OPN   DB [#WT_DB];
      T     %DBW68;  //"DB_WT1".Speed_Fahrt
      L     "DB_Techno".KorrPend;  //Korrektur Pendeln laden
      OPN   DB [#WT_DB];
      T     %DBD38;
      L     "DB_Techno".KorrATZ;  //Korrektur Tropfen laden
      OPN   DB [#WT_DB];
      T     %DBD42;
      L     "DB_Techno".WT_Kennung;
      OPN   DB [#WT_DB];
      T     %DBB63;
      L     "DB_Techno".WT_Typ;
      OPN   DB [#WT_DB];
      T     %DBB35;

      OPN   DB [#WT_DB];
      A     #WT_nok;  //nok zurückladen
      =     %DBX22.3;  //"DB_WT1".WT_nok

      CALL  "FC_TechScan"
      ( WT_DB_Nr := #WT_DB
      );

      AN    #WTnew;
      JC    OEvt;
//------------------------
//Daten bei neuem WT
//------------------------

      L     "DB_Techno".Oberflaeche;
      OPN   DB [#WT_DB];
      T     %DBD10;
      L     0;
      T     %DBW46;  //Parameterpointer
      T     %DBW48;  //Befehlspointer
      T     %DBB20;  //Behandlungsbits
      T     %DBD30;  //"DB_WT1".Fertigzeitpunkt

      L     "DB_Techno".Korb_Nr;
      OPN   DB [#WT_DB];
      T     %DBB14;  //"DB_WTx".Korb_Nr

      CALL  "FC_Korbumlaeufe"
      ( Nr := "DB_Techno".Korb_Nr
      );

      L     "DB_Techno".Technologie;
      OPN   DB [#WT_DB];
      T     %DBW16;  //Technologienummer
      OPN   DB [#WT_DB];
      L     #Pos_Nr;
      T     %DBB15;  //WT Ist-Pos
      T     %DBB19;  //WT Auto-Pos

      L     "DB_Panel_OVERVIEW".Systime;
      OPN   DB [#WT_DB];
      T     %DBD74;  //"DB_WT1".Aufgabezeit

      SET;
      R     %DBX20.0;  //Trommel
      S     %DBX18.1;  //in Anlage
      R     %DBX18.2;  //in Entmetallisierung
      R     %DBX18.3;  //aus Anlage
      R     %DBX18.4;  //aus Entmetallisierung
      R     %DBX18.5;  //Speicherprogramm


NETWORK
TITLE = 
// WT in Position laden
      CALL  "FC_WT_to_Pos"
      ( Pos_Nr     := #Pos_Nr,
        WT_Nr      := #WT_Nr,
        BA_Auto    := TRUE,
        send_DBEvt := FALSE,
        SimLoad    := FALSE,
        Copy_ok    := #"Return"
      );

// Langware in beide Positionen laden

      L     "DB_Techno".WT_Typ;
      L     b#16#12;  //Lang schmal
      <>I;
      JC    ende;
      L     #Pos_Nr;
      INC   1;
      T     #Pos_Nr;

      CALL  "FC_WT_to_Pos"
      ( Pos_Nr     := #Pos_Nr,
        WT_Nr      := #WT_Nr,
        BA_Auto    := TRUE,
        send_DBEvt := FALSE,
        SimLoad    := FALSE,
        Copy_ok    := #"Return"
      );

      JU    ende;

OEvt: NOP   0;

      CALL  "FC_WT_from_Pos"
      ( Pos_Nr     := #Pos_Nr,
        send_DBEvt := FALSE,
        load_ok    := #"Return",
        WT_Nr      := #WT_kurz,
        WT_Nr_lang := #WT_lang
      );

      AN    #"Return";
      JC    ende;

      CALL  "FC_WT_to_Pos"
      ( Pos_Nr     := #Pos_Nr,
        WT_Nr      := #WT_kurz,
        BA_Auto    := FALSE,
        send_DBEvt := FALSE,
        SimLoad    := FALSE,
        Copy_ok    := #"Return"
      );

ende: BE;

END_FUNCTION

FUNCTION "FC_DB_COPY" : Void   // FC3, STL
TITLE = Blocktransfer
{ S7_Optimized_Access := 'FALSE' }
AUTHOR : MS
// Kopiert Datenblöcke von Quell- zu Ziel-DB und löscht(bei CLR_ALT_DB) 
// anschließend eingetragenen Bereich im Quell-Db
// stored: AutoNumber false
   VAR_INPUT
      CLR_ALT_DB : Bool;   // NACH DEM KOPIEREN WIRD DER URSPRUNG-DB GELÖSCHT
      ALT_DB : Int;   // URSPRUNG DB
      NEU_DB : Int;   // ZIEL DB
      COPY_START : Int;   // ADRESSE DES WORTES, WELCHES ALS ERSTES KOPIERT WIRD
      COPY_ENDE : Int;   // ADRESSE DES WORTES, WELCHES ALS ERSTES NICHT MEHR KOPIERT WIRD
      ZIEL_START : Int;   // STARTADRESSE DATENBEREICH ZIEL
      CLR_START : Int;   // ADRESSE DES WORTES, WELCHES ALS ERSTES GELÖSCHT WIRD
      CLR_ENDE : Int;   // ADRESSE DES WORTES, WELCHES ALS ERSTES NICHT MEHR GELÖSCHT WIRD
   END_VAR
   VAR_IN_OUT
      START : Bool;   // DURCHLAUFMERKER/OK-SIGNAL
   END_VAR
   VAR_TEMP
      ZAEHLER1 : Int;   // ZAEHLVARIABLE QUELLE
      ZAEHLER2 : Int;   // ZAEHLVARIABLE ZIEL
      Alt_DB1 : Word;
      Neu_DB1 : Word;
   END_VAR
BEGIN

NETWORK
TITLE = Copy
// DATENBEREICH KOPIEREN
      L     #ALT_DB;
      T     #Alt_DB1;
      OPN   DI [#Alt_DB1];
      L     #NEU_DB;
      T     #Neu_DB1;
      OPN   DB [#Neu_DB1];
      AN    #START;
      BEC;
      L     #COPY_START;
      T     #ZAEHLER1;
      L     #ZIEL_START;
      T     #ZAEHLER2;
COPY: L     #ZAEHLER1;
      SLD   3;
      LAR1;
      L     #ZAEHLER2;
      SLD   3;
      LAR2;
      L     DIW [AR1, P#0.0];
      T     DBW [AR2, P#0.0];
      L     #ZAEHLER2;
      L     2;
      +D;
      T     #ZAEHLER2;
      L     #ZAEHLER1;
      L     2;
      +D;
      T     #ZAEHLER1;
      L     #COPY_ENDE;
      <I;
      JC    COPY;

NETWORK
TITLE = Delete
// DATENBEREICH DER QUELLE MIT "0" FÜLLEN
      AN    #CLR_ALT_DB;
      JC    AUS;
      L     #CLR_START;  //STARTADRESSE WORT LÖSCHEN
      T     #ZAEHLER1;
DEL:  L     #ZAEHLER1;
      SLD   3;
      LAR1;
      L     0;
      T     DIW [AR1, P#0.0];
      L     #ZAEHLER1;
      L     2;
      +D;
      T     #ZAEHLER1;
      L     #CLR_ENDE;  //ENDADRESSE WORT LÖSCHEN
      <I;
      JC    DEL;

NETWORK
TITLE = Ready
// ENDE /FERTIGMELDUNG
AUS:  CLR;
      =     #START;
      BE;
END_FUNCTION

FUNCTION "FC_TechScan" : Void   // FC42, STL
TITLE = Initialisieren Technologische Parameter
{ S7_Optimized_Access := 'FALSE' }
// stored: AutoNumber false
   VAR_INPUT
      WT_DB_Nr : Int;
   END_VAR
   VAR_TEMP
      WT_DB : Word;
      lastCmd : Int;
      Count : Int;
      AdrReg1 : DWord;
      AdrReg2 : DWord;
      typTaktzeit : Int;
      Expo : DInt;
   END_VAR
BEGIN

NETWORK
TITLE = Bereichstakte Beladestand 1 laden

//-------------------------------
//WT-DB öffnen und Adressregister
//retten
//-------------------------------
      TAR1;
      T     #AdrReg1;
      TAR2;
      T     #AdrReg2;

      L     "DB_ANLAGE".config.Taktzeit_typ;
      T     #typTaktzeit;

      L     #WT_DB_Nr;
      T     #WT_DB;
      OPN   DB [#WT_DB];

//-------------------------------
//Initialisieren Kopfdaten
//-------------------------------
      L     0;
      T     %DBB54;  //"DB_WT1".Variante0//Bereichstakte
      T     %DBB55;  //"DB_WT1".Variante1  Technologie 0=Natur, 1=Matt, 2=Glänzen
      T     %DBB56;  //"DB_WT1".Variante2  Farbe 0-6
      T     %DBB57;  //"DB_WT1".Variante3  Beizzeit 0=<60s 1=<8min 2=>8min
      T     %DBB58;  //"DB_WT1".Variante4  Glänzzeit 0=kurz 1=mittel 2=lang
      T     %DBB59;  //"DB_WT1".Variante5


NETWORK
TITLE = Scan Technologie
//-------------------------------
//Scan von Befehl 0 bis Anzahl
//-------------------------------
      L     %DBW0;  //"DB_WT1".ANZAHL
      T     #lastCmd;
      L     0;
retC: T     #Count;
      L     #lastCmd;
      >=I;
      JC    Ende;

      L     #Count;
      L     %DBW4;  //"DB_WT1".LENG
      *I;
      L     %DBW2;  //"DB_WT1".OFFSET
      +I;
      SLD   3;
      LAR1;
      OPN   DB [#WT_DB];
      L     DBB [AR1, P#0.0];  //CmdID
      L     0;
      ==I;
      JC    Ende;

nexC: L     #Count;
      +     1;
      JU    retC;

NETWORK
TITLE = Parameter abfregen und laden

NETWORK
TITLE = Ende Scandurchlauf
Ende: L     #AdrReg1;
      LAR1;
      L     #AdrReg2;
      LAR2;
      BE;
END_FUNCTION

FUNCTION "FC_Korbumlaeufe" : Void   // FC330, LAD
TITLE = Korbumläufe
{ S7_Optimized_Access := 'TRUE' }
// stored: AutoNumber false, SetENOAutomatically false
   VAR_INPUT
      Nr : USInt;
   END_VAR
BEGIN

REGION Network 1 (SCL): Check Korb-Nr
   IF (#Nr < "KorbAnzahl_min") OR (#Nr > "KorbAnzahl_max") THEN
       RETURN;
   END_IF;
END_REGION

REGION Network 2 (SCL): Zählen und Maxwert checken
   "DB_Korbumlaeufe".Korb[#Nr].Durchlaeufe := "DB_Korbumlaeufe".Korb[#Nr].Durchlaeufe + 1;
END_REGION
END_FUNCTION

FUNCTION "FC_WT_to_Pos" : Void   // FC51, STL
TITLE = Laden von WT-Daten in eine Position
{ S7_Optimized_Access := 'FALSE' }
// Wird beim Einsetzen eines WT in eine Position ausgeführt.
// Aufruf durch Transportwagen und Quertransporte sowie auf Beladeständen
// stored: AutoNumber false
   VAR_INPUT
      Pos_Nr : USInt;   // Positionsnummer in die der WT geladen wird
      WT_Nr : Byte;   // Nr. des Warenträgers, der in die Position geladen werden soll.
      BA_Auto : Bool;   // Umladen erfolgt in der Betriebsart Automatik
      send_DBEvt : Bool;   // Datenbank-Events senden
      SimLoad : Bool;   // WT-laden wird simuliert damit richtige Einstellungen im Bad
   END_VAR
   VAR_OUTPUT
      Copy_ok : Bool;   // Kopiervorgang erfolgreich abgeschlossen
   END_VAR
   VAR_TEMP
      WT_NR_LANG : DInt;
      WT_lang : DWord;
      Param : DWord;
      Summ_Temp : Real;
      WT_DB : Word;   // Datenbaustein mit Warenträgerinformationen
      Pntr_ret : Int;
      akt_Bef_Nr : Int;
      Ziel_1 : Byte;
      Ziel_2 : Byte;
      Ziel_x : Byte;
      Ziel_y : Byte;
      leng_1 : Byte;
      leng_2 : Byte;
      P_fnd : Bool;
      not_load : Bool;   // WT nicht umladen!!!
      WT_Neuaufgabe : Bool;   // WT wurde neu aufgegeben (keine Index-Korrektur)
      group_load : Bool;
      Auto : Bool;
   END_VAR
BEGIN

NETWORK
TITLE = Initialisierung und Gültigkeitsprüfung
//---------------------------
//Initialisieren
//---------------------------
      SET;
      R     #Copy_ok;
      A     #BA_Auto;
      =     #Auto;
//---------------------------
//WT_DB ermitteln
//---------------------------
      L     0;
      L     #WT_Nr;
      >=I;
      BEC;
      L     100;
      +I;
      T     #WT_DB;
//---------------------------
//Adressregister Pos. laden
//---------------------------
      L     "DB_ANLAGE".config.ANZ_Pos;
      L     #Pos_Nr;
      <I;
      BEC;
      L     0;
      <=I;
      BEC;

      CALL  "FC_POS_TO_WORK"
      ( Akt_Pos  := #Pos_Nr,
        not_load := #not_load
      );
      A     #not_load;
      BEC;
//---------------------------
//Pos. bereits belegt
//---------------------------
      L     "DB_POS".POS[0].WT_DB;
      L     0;
      <>I;
      AN(;
      L     "DB_POS".POS[0].WT_DB;
      L     #WT_Nr;
      ==I;
      );
      BEC;


NETWORK
TITLE = Ladevorgang

      OPN   DB [#WT_DB];
      L     %DBD6;  //WT_Nr_lang
      T     #WT_NR_LANG;

      AN    #send_DBEvt;
      O     #SimLoad;
      JC    noDB;

//----------------------------
//Parameteradresse prüfen
//und Parameter umladen
//----------------------------
noDB: A     #Auto;
      JC    ok;
      OPN   DB [#WT_DB];
      R     %DBX20.5;  //"DB_WT1".noKorrBefx

      L     0;
      T     %DBB36;  //"DB_WT1".End_Ziel_Pos
      T     %DBB37;  //"DB_WT1".End_Ziel_Reihe

ok:   OPN   DB [#WT_DB];
      L     %DBW48;  //Befehl-Nr
      T     #akt_Bef_Nr;

//WT wurde neu aufgegeben --> Befehlsindex nicht weiterschalten
      L     "DB_POS".POS[0].Stand_Nr;
      L     0;
      <>I;
      A(;
      OPN   DB [#WT_DB];
      L     %DBW48;  //Befehlsindex
      L     0;
      ==I;
      );
      O(;
      OPN   DB [#WT_DB];
      L     %DBD6;  //"DB_WT1".WT_NR_lang
      L     0;
      ==D;
      );
      =     #WT_Neuaufgabe;
      =     #P_fnd;
      JC    noPa;

// Bei Langware und gerader Position nichts tun!!
      L     #Pos_Nr;
      L     2;
      MOD;
      A     ==0;  // gerade
      A(;
      OPN   DB [#WT_DB];
      L     %DBB35;  //"DB_WTx".WT_Typ
      L     "WT_Typ_LS";
      ==I;
      );
      R     #P_fnd;
      JC    noPa;

//WT erreicht Endziel eines komplexen Umsetzvorganges (Gruppe bzw. F_Posfree)
      OPN   DB [#WT_DB];
      L     0;
      L     %DBB36;  //"DB_WT1".End_Ziel_Pos
      ==I;
      JC    SPos;  //WT Sondertransport

      L     #Pos_Nr;
      L     %DBB36;  //"DB_WT1".End_Ziel_Pos
      ==I;
      JC    ZpEr;

      L     %DBW48;  //Befehlsindex
      L     %DBW4;  //Länge
      *I;
      L     %DBW2;  //Offset
      +I;
      SLD   3;
      LAR1;
      L     DBB [AR1, P#1.0];  //Ziel-Basispos
      T     #Ziel_1;
      L     DBB [AR1, P#2.0];  //Ziel-Länge
      +I;
      +     -1;
      T     #Ziel_x;

      L     DBB [AR1, P#3.0];  //Ziel-Basispos
      T     #Ziel_2;
      L     DBB [AR1, P#4.0];  //Ziel-Länge
      +I;
      +     -1;
      T     #Ziel_y;

//DBB36 in erstem Gruppenabschnitt?
      L     #Ziel_1;
      L     0;
      ==I;
      JC    SPos;
      L     %DBB36;  //"DB_WT1".End_Ziel_Pos
      L     #Ziel_1;
      <I;
      O(;
      L     %DBB36;  //"DB_WT1".End_Ziel_Pos
      L     #Ziel_x;
      >I;
      );
      JC    chk2;
//IstPosition in erstem Gruppenabschnitt?
      L     #Pos_Nr;
      L     #Ziel_1;
      <I;
      O(;
      L     #Pos_Nr;
      L     #Ziel_x;
      >I;
      );
      JC    chk2;
      JU    ZpEr;

//DBB36 in zweitem Gruppenabschnitt?
chk2: L     #Ziel_2;
      L     0;
      ==I;
      JC    SPos;
      L     %DBB36;  //"DB_WT1".End_Ziel_Pos
      L     #Ziel_2;
      <I;
      O(;
      L     %DBB36;  //"DB_WT1".End_Ziel_Pos
      L     #Ziel_y;
      >I;
      );
      JC    SPos;
//IstPosition in zweitem Gruppenabschnitt?
      L     #Pos_Nr;
      L     #Ziel_2;
      <I;
      O(;
      L     #Pos_Nr;
      L     #Ziel_y;
      >I;
      );
      JC    SPos;

ZpEr: SET;
      R     %DBX20.5;
      L     0;
      T     %DBB36;
      T     %DBB37;

SPos: SET;
      R     #group_load;

      A     %DBX20.5;
      R     #P_fnd;
      JC    noPa;

      CALL  "FC_Pointer_Tech"
      ( Befehl       := #akt_Bef_Nr,
        Position     := #Pos_Nr,
        WT_Nr        := #WT_DB,
        p_fnd        := #P_fnd,
        new_Bef_Pntr := #Pntr_ret
      );  //Adresse prüfen und korregieren

      AN    #P_fnd;  //keine gültige Adresse gefunden
      JC    noPa;

      OPN   DB [#WT_DB];  //Pointer für Parameter übernehmen
      L     #Pntr_ret;
      T     %DBW48;

      CALL  "FC_PAR_COPY"
      ( Pos_Nr   := #Pos_Nr,
        WT_DB_Nr := #WT_DB
      );  //Parameter ins Bad laden

//-------------------------------------------
// Umsetzvorgang innerhalb einer Gruppe?
//-------------------------------------------
      OPN   DB [#WT_DB];
      L     #Pos_Nr;
      L     %DBB19;  //"DB_WT1".Auto_Pos
      ==I;
      ON    "DB_POS".POS[0].enable_reload;
      JC    noPa;

      OPN   DB [#WT_DB];
      L     %DBW48;  //Befehlsindex
      L     %DBW4;  //Länge
      *I;
      L     %DBW2;  //Offset
      +I;
      SLD   3;
      LAR1;
      L     DBB [AR1, P#1.0];  //Ziel-Basispos
      T     #Ziel_1;
      L     DBB [AR1, P#2.0];  //Ziel-Länge
      +I;
      L     1;
      -I;
      JM    noPa;
      T     #Ziel_x;

      L     #Ziel_1;
      L     %DBB19;  //"DB_WT1".Auto_Pos
      <=I;
      A(;
      L     #Ziel_x;
      <=I;
      );
      =     #group_load;
      JC    noPa;

      L     DBB [AR1, P#3.0];  //Ziel-Basispos
      T     #Ziel_2;
      L     DBB [AR1, P#4.0];  //Ziel-Länge
      +I;
      L     1;
      -I;
      JM    noPa;
      T     #Ziel_y;

      L     #Ziel_2;
      L     %DBB19;  //"DB_WT1".Auto_Pos
      <=I;
      A(;
      L     #Ziel_y;
      <=I;
      );
      =     #group_load;


NETWORK
TITLE = Position aktualisieren
//----------------------------
//WT in Pos laden
//----------------------------
noPa: SET;
      S     #Copy_ok;
      AN    #SimLoad;
      JC    norm;

      OPN   DB [#WT_DB];
      A     %DBX20.0;  //Trommel
      =     "DB_POS".POS[0].Trommel;
      OPN   DB [#WT_DB];
      L     %DBD10;  //Oberfläche
      T     "DB_POS".POS[0].KF_A;
      L     0.0;
      ==R;
      =     "DB_POS".POS[0].Leer_WT;
      JU    SimL;

norm: S     "DB_POS".POS[0].belegt;
      A     #send_DBEvt;
      S     "DB_POS".POS[0].WT_neu;

      OPN   DB [#WT_DB];
      L     "WT_Typ_KS";
      L     %DBB35;  //WT-Typ
      ==I;
      =     "DB_POS".POS[0].Belegt_KS;
      L     "WT_Typ_LS";
      ==I;
      =     "DB_POS".POS[0].Belegt_LS;
      CAC;
      L     "WT_Typ_GO";
      ==I;
      =     "DB_POS".POS[0].Belegt_GO;

      L     #WT_Nr;
      T     "DB_POS".POS[0].WT_DB;
      T     "DB_POS".POS[0].next_WT;

      L     #WT_NR_LANG;
      T     "DB_POS".POS[0].WT_Nr_lang;

//-------------------------------
//WT Befehlsindex überprüfen
//-------------------------------
      OPN   DB [#WT_DB];
      A     #send_DBEvt;
      R     %DBX20.2;  //Stop gefordert

//Befehlsindex weiter schalten
      A     #WT_Neuaufgabe;
      ON    "DB_POS".POS[0].Bef_ende;  //kein Bef. schalten erforderlich
      JC    GET;

      OPN   DB [#WT_DB];
      L     %DBW48;  //Befehlsindex
      L     %DBW4;  //Länge
      *I;
      L     %DBW2;  //Offset
      +I;
      SLD   3;
      LAR1;

      A     #P_fnd;  //ungültiger Befehlszeiger
      JC    newX;
//-----------------------------
//Prüfung ob WT hier richtig
//-----------------------------
      L     DBB [AR1, P#0.0];  //Command-ID
      L     16#F0;  //Einfahrt über freien Weg zur Optipos
      ==I;
      A     "DB_POS".POS[0].Optipos;
      JC    newX;
      JU    chkS;

newX: OPN   DB [#WT_DB];
      L     %DBW48;  //Befehlsindex erhöhen
      L     1;
      +I;
      T     %DBW48;

      L     %DBW4;  //Länge
      *I;
      L     %DBW2;  //Offset
      +I;
      SLD   3;
      LAR1;  //Adresse neuer Befehl

chkS: OPN   DB [#WT_DB];
      L     DBB [AR1, P#0.0];  //Command-ID
      L     16#FF;  //Trockneranforderung
      ==I;
      S     %DBX20.1;  //Trockneranforderung
      JC    newX;

      L     DBB [AR1, P#0.0];  //Command-ID
      L     16#FE;  //Stopbefehl
      ==I;
      S     %DBX20.2;  //Stop aktiv
      JC    newX;

GET:  OPN   DB [#WT_DB];
      A     %DBX20.0;  //Trommel
      =     "DB_POS".POS[0].Trommel;
      OPN   DB [#WT_DB];
      L     %DBD10;  //Oberfläche
      T     "DB_POS".POS[0].KF_A;
      L     0.0;
      ==R;
      =     "DB_POS".POS[0].Leer_WT;

      OPN   DB [#WT_DB];
      L     %DBB14;  //WT_Nr kurz
      T     "DB_POS".POS[0].WT_Stangen_Nr;
      OPN   DB [#WT_DB];
      L     %DBW48;  //Befehlsindex
      T     "DB_POS".POS[0].WT_Befx;

      L     "DB_POS".POS[0].SubTyp;
      L     1;
      ==I;
      OPN   DB [#WT_DB];
      AN    %DBX18.1;  //in die Anlage
      JC    nMem;

      L     "DB_POS".POS[0].Typ;
      L     5;  //Speicher
      <>I;
      JC    nMem;

      OPN   DB [#WT_DB];
      AN    %DBX22.3;  //"DB_WT1".WT_nok
      JC    WTok;

WTok: OPN   DB [#WT_DB];
      L     %DBW2;  //"DB_WT1".OFFSET
      SLD   3;
      LAR1;
      L     DBB [AR1, P#0.0];  //Befehl Speicherprogramm?
      L     16#FA;  //250
      ==I;
      O     %DBX18.5;  //"DB_WT1".Speicher
      S     "DB_POS".POS[0].Sperre_out;

nMem: A     "DB_POS".POS[0].Optipos;
      JC    OptE;

//Bereichstakte aus Pos übernehmen
      L     0;
      L     "DB_POS".POS[0].BereichsTakte;
      ==I;
      JC    nBT;
      OPN   DB [#WT_DB];
      T     %DBB54;  //"DB_WT1".Bereichstakte

nBT:  L     "DB_POS".POS[0].Soll_Takte;
      T     "DB_POS".POS[0].Resttakte;
      L     0;
      ==I;
      JC    noKo;
      L     "DB_POS".POS[0].Soll_Takte;
      L     "DB_ANLAGE".config.Taktzeit_typ;
      *D;
      T     "DB_POS".POS[0].Soll_Expozeit;

noKo: L     "DB_POS".POS[0].Soll_Expozeit;
      DTR;
      L     "DB_POS".POS[0].KF_Expo;
      *R;
      RND+;
      T     "DB_POS".POS[0].Restzeit;
      JU    GO;

//--------------------------------------
//Optimierungsrechnung anfordern WT-Neu
//--------------------------------------
OptE: NOP   0;

//--------------------------------------
//Positionsdaten zurückladen
//--------------------------------------
GO:   SET;
      S     "DB_POS".POS[0].Bearbeitung;
      L     "DB_POS".POS[0].KF_A;
      L     0.0;
      ==R;
      =     "DB_POS".POS[0].Leer_WT;

      OPN   DB [#WT_DB];
      L     %DBB18;
      OPN   "DB_POS";
      T     %DBB87;  //  "DB_POS".POS[0].Speicherbits

      L     "DB_POS".POS[0].Typ;
      L     5;
      <>I;
      AN    "DB_POS".POS[0].Optipos;
      JC    ndST;
      OPN   DB [#WT_DB];
      L     0;
      T     %DBD50;  //"DB_WT1".SaveExpo

ndST: OPN   DB [#WT_DB];
      SET;
      R     %DBX20.4;  //"DB_WT1".TW_Pos

      L     #Pos_Nr;
      OPN   DB [#WT_DB];
      T     %DBB15;  //POSITION

      OPN   DB [#WT_DB];
      L     %DBB21;  //gemerkte Ziel-Position
      L     #Pos_Nr;
      ==I;
      S     #Auto;  //letzter Umsetzvorgang in Automatik

      AN    #Auto;
      AN    #group_load;
      R     %DBX20.7;  //"DB_WT1".last_Auto
      JC    nAu;
      AN    #group_load;
      JC    nAu;
      S     %DBX20.7;  //"DB_WT1".last_Auto

      L     #Pos_Nr;
      T     %DBB19;  //AUTOPOSITION

nAu:  OPN   DB [#WT_DB];  //Wird gerade abgeholt
      A     %DBX18.1;  //"DB_WT1".in_Anlage
      O     %DBX18.2;  //"DB_WT1".in_Entm
      A     "DB_POS".POS[0].Optipos;
      A     "DB_POS".POS[0].Quelle;
      JC    OptP;

      L     "DB_POS".POS[0].Typ;
      JL    Tlst;
      JU    Anl;  //Anlagenbad
      JU    end3;  //Beladen
      JU    end3;  //Entladen
      JU    end3;  //Be- und Entladen
      JU    end3;  //frei
      JU    end3;  //Speicher
Tlst: JU    end3;

Anl:  OPN   DB [#WT_DB];
      L     %DBB15;  //ALTPOSITION IM AUTO
      L     %DBB19;  //AUTOPOSITION
      <>I;
      JC    end3;

      L     "DB_POS".POS[0].SubTyp;  //Werte zurückladen auch in Automatik
      L     5;
      <>I;
      A     #Auto;  //letzter Umsetzvorgang in Automatik
      AN    #group_load;
      JC    end3;

OptP: OPN   DB [#WT_DB];
      L     %DBB24;  //"DB_WT1".Alt_Bereichstakte
      T     %DBB54;  //"DB_WT1".Bereichstakte

      A     %DBX25.0;  //"DB_WT1".Alt_TW_Pos
      =     %DBX20.4;  //"DB_WT1".TW_Pos

      OPN   DB [#WT_DB];
      L     %DBD26;  //ALT VERWEILZEIT
      T     "DB_POS".POS[0].Verweilzeit;
      OPN   DB [#WT_DB];
      L     %DBB23;  //Befehlsindex
      T     %DBW48;
      T     "DB_POS".POS[0].WT_Befx;
      OPN   DB [#WT_DB];
      AN    #group_load;
      JC    setA;
      L     0;
      T     %DBD50;  //"DB_WT1".SaveExpo
setA: SET;
      =     #Auto;  //letzter Umsetzvorgang in Automatik


NETWORK
TITLE = Normale Badbehandlung
// Aufruf der allgemeinen Badbehandlung
end3: AN    #Auto;
      JC    noAu;
      OPN   DB [#WT_DB];
      S     %DBX20.7;  //"DB_WT1".last_Auto

      L     #Pos_Nr;
      T     %DBB19;  //AUTOPOSITION

noAu: NOP   0;

      CALL  "FC_Pos_Behandlung"
      ( Pos_Nr     := #Pos_Nr,
        send_DBEvt := #send_DBEvt
      );
//-------------------------------
//zurückladen der PosDaten
//-------------------------------
SimL: CALL  "FC_WORK_TO_POS"
      ( Akt_Pos := #Pos_Nr
      );

END_FUNCTION

FUNCTION "FC_POS_TO_WORK" : Void   // FC53, STL
TITLE = Arbeitsdaten einlesen
{ S7_Optimized_Access := 'FALSE' }
AUTHOR : MS
// Überträgt die Positionsdaten zur Bearbeitung in den Bearbeitungs-DB
// stored: AutoNumber false
   VAR_INPUT
      Akt_Pos : USInt;   // Position die geladen wird
   END_VAR
   VAR_OUTPUT
      not_load : Bool;   // Position nicht laden
   END_VAR
BEGIN

NETWORK
TITLE = Copy Data
// Lädt Daten der aktuellen Position in Feld [0]
      L     "DB_POS".POS[#Akt_Pos].Typ;
      L     B#16#FF;
      ==I;
      =     #not_load;
      BEC;

      CALL  MOVE
      ( IN  := "DB_POS".POS[#Akt_Pos],
        OUT := "DB_POS".POS[0]
      );

END_FUNCTION

FUNCTION "FC_Pointer_Tech" : Void   // FC16, STL
TITLE = Pointer setzen
{ S7_Optimized_Access := 'FALSE' }
AUTHOR : MS
// aktualisiert Befehlsnummer des WT
// stored: AutoNumber false
   VAR_INPUT
      Befehl : Int;
      Position : USInt;
      WT_Nr : Word;
   END_VAR
   VAR_OUTPUT
      p_fnd : Bool;   // gültigen Parameter gefunden
      new_Bef_Pntr : Int;   // neuer Befehlspointer
   END_VAR
   VAR_TEMP
      Bef1 : Int;
      QT_DB : Int;
      Abstand1 : Int;
      Abstand2 : Int;
      Anzahl_B : Int;   // Anzahl der Befehle
      Laenge_B : Int;   // Länge eines Befehls
      start_adr : Word;
      Offset : Word;
      WT_DB : Word;
      akt_Pos : Byte;
      Ziel1 : Byte;
      leng1 : Byte;
      Ziel2 : Byte;
      leng2 : Byte;
      GroupNr : Byte;
      firstChk : Bool;
      temp_p_fnd : Bool;
   END_VAR
BEGIN

NETWORK
TITLE = search TechNr
// Technologie-Munner im Inhaltsverzeichnis suchen und Offset ermitteln
//------------------------
//Initialisieren
//------------------------
      L     0;
      T     #Bef1;
      T     #Abstand1;
      T     #Abstand2;
      T     #new_Bef_Pntr;
      T     #start_adr;

      SET;
      S     #firstChk;
      R     #temp_p_fnd;


NETWORK
TITLE = scan Bef_Nr
// scannen ob für dei aktuelle Position Einträge existieren
// bis zu 3 Einträge werden übernommen
//------------------------
//Initialisieren
//------------------------
      L     #WT_Nr;
      T     #WT_DB;
      OPN   DB [#WT_DB];
      L     %DBW0;  //Anzahl Befehle
      T     #Anzahl_B;
      L     %DBW2;  //Offset
      T     #Offset;
      L     %DBW4;  //Länge
      T     #Laenge_B;

//-------------------------
//Befehl passt bereits
//aktueller Pointer prüfen
//-------------------------
      L     #Befehl;
      L     #Laenge_B;
      *I;
      L     #Offset;
      +I;
      SLD   3;
      LAR1;
      JU    Chk;

//------------------------
//Eintrag prüfen
//------------------------
such: A     #firstChk;
      R     #firstChk;
      JC    nexB;
      L     #start_adr;
      +     1;
      T     #start_adr;
      L     #Anzahl_B;
      >=I;
      JC    ende;

nexB: L     #start_adr;
      L     #Laenge_B;
      *I;
      L     #Offset;
      +I;
      SLD   3;
      LAR1;
      JU    Chk;

//------------------------
//Eintrag gefunden
//------------------------
fnd:  A     #firstChk;
      R     #firstChk;
      S     #temp_p_fnd;
      JC    raus;

      AN    #temp_p_fnd;  //erster gefundener Eintrag
      S     #temp_p_fnd;
      JC    take;

//------------------------
//Eintrag vergleich/merken
//------------------------
      L     #Bef1;
      L     #Befehl;
      -I;
      ITD;
      DTR;
      ABS;
      RND;
      T     #Abstand1;

      L     #start_adr;
      L     #Befehl;
      -I;
      ITD;
      DTR;
      ABS;
      RND;
      T     #Abstand2;

      L     #Abstand1;
      L     #Abstand2;
      <I;
      JC    such;
take: L     #start_adr;
      T     #Bef1;
      JU    such;


NETWORK
TITLE = Prüfe Befehl
//----------------------------------------------------------------------
//ungültig
Chk:  OPN   DB [#WT_DB];
      L     0;  //Ende Suchbereich
      L     DBB [AR1, P#0.0];  //"DB_WT1".Befehl[0].Kennung
      ==I;
      JCN   prf;
      AN    #firstChk;
      JC    ende;
      JU    such;  //nichts gefunden --> Technologie scannen!

//240-249 (F0..F9) Gruppenfahrt
prf:  L     249;  //Ende Suchbereich
      L     DBB [AR1, P#0.0];  //"DB_WT1".Befehl[0].Kennung
      >=I;
      A(;
      L     240;  //Ende Suchbereich
      >=I;
      );
      JC    Grp;  //nichts gefunden --> Technologie scannen!

//230-235 (E6..EB) Quertransport
      L     235;
      L     DBB [AR1, P#0.0];  //Kennung
      >=I;
      A(;
      L     230;
      >I;
      );
      JC    QT;  //QT-Befehl

//254 (FE) Kontrolle//Sonderbefehle überspringen
//255 (FF) Trockner einschalten
      L     DBB [AR1, P#0.0];  //Cmd
      L     254;
      >I;
      JC    such;

//bis 220 normal
//220-229 (DC..E5) Variante --> normal
//250-252 (FA..FC) Speicherfahrt --> normal
      JU    Norm;
//----------------------------------------------------------------------



//----------------------------------------------------------------------
//Normalbefehl
Norm: OPN   DB [#WT_DB];
      L     0;
      L     DBB [AR1, P#1.0];  //Posangabe
      ==I;
      JC    such;
      L     DBB [AR1, P#1.0];  //Posangabe
      T     #Ziel1;
      L     DBB [AR1, P#2.0];  //Länge der Badgruppe
      T     #leng1;
      L     DBB [AR1, P#3.0];  //Posangabe
      T     #Ziel2;
      L     DBB [AR1, P#4.0];  //Länge der Badgruppe
      T     #leng2;

nxL:  L     #leng1;
reP:  T     #leng1;
      L     1;
      -I;
      L     #Ziel1;
      +I;
      T     #akt_Pos;

      L     #akt_Pos;
      L     #Position;
      ==I;
      JC    fnd;

      L     #leng1;
      LOOP  reP;

      L     #Ziel2;
      L     0;
      ==I;
      JC    such;
      L     #Ziel2;
      T     #Ziel1;
      L     #leng2;
      T     #leng1;
      L     0;
      T     #Ziel2;
      T     #leng2;
      JU    nxL;
//----------------------------------------------------------------------
//----------------------------------------------------------------------
//QT-Befehl prüfen
QT:   -I;
      L     5;
      >I;
      JC    such;
      CAC;
      +     30;
      T     #QT_DB;
      OPN   DB [#QT_DB];
      L     #Position;
      L     %DBB60;  //"DI_QT_1".PAR.POS1
      ==I;
      JC    fnd;
      L     #Position;
      L     %DBB61;  //"DI_QT_1".PAR.POS2
      ==I;
      JC    fnd;
      L     #Position;
      L     %DBB62;  //"DI_QT_1".PAR.POS3
      ==I;
      JC    fnd;
      L     #Position;
      L     %DBB63;  //"DI_QT_1".PAR.POS4
      ==I;
      JC    fnd;
      L     #Position;
      L     %DBB64;  //"DI_QT_1".PAR.POS5
      ==I;
      JC    fnd;
      JU    such;
//----------------------------------------------------------------------
//----------------------------------------------------------------------
//nach Gruppe suchen
Grp:  -I;
      T     #GroupNr;
      L     9;
      <=I;
      JCN   such;

//------------------------
//Eintrag prüfen
//------------------------
      L     #GroupNr;
      L     "DB_GroupConfig".AnzGroup;
      >=I;
      JC    such;

//--------------------------------------
//Gruppe öffnen
//--------------------------------------
      L     #GroupNr;
      L     6;
      *D;
      L     "DB_GroupConfig".OffsetAdr;
      +D;
      SLD   3;
      LAR1;
      OPN   "DB_GroupConfig";
//--------------------------------------
//Eintragsadresse berechnen
//--------------------------------------
      L     DBW [AR1, P#0.0];  //"DB_GroupConfig".Gruppe[0].Start
      SLD   3;
      LAR1;
retP: OPN   "DB_GroupConfig";
//--------------------------------------
//letzter Gruppeneintrag gefunden
//--------------------------------------
      L     0;
      L     DBB [AR1, P#0.0];
      ==I;
      JC    such;
      L     #Position;
      ==I;
      JC    fnd;
//--------------------------------------
//nächste Position
//--------------------------------------
      +AR1  P#1.0;
      JU    retP;
//----------------------------------------------------------------------


NETWORK
TITLE = Auswertung
ende: NOP   0;
//------------------------
//kein Eintrag?
//------------------------
      AN    #temp_p_fnd;
      JC    Out;  //   BEB
//----------------------------
//Eitrag übernehmen
//----------------------------
      L     #Bef1;
      T     #new_Bef_Pntr;
      JU    Out;  //    BE

raus: L     #Befehl;
      T     #new_Bef_Pntr;
      JU    Out;  //  BE

//Outputvariablen Umkopieren
Out:  A     #temp_p_fnd;
      =     #p_fnd;
END_FUNCTION

FUNCTION "FC_PAR_COPY" : Void   // FC55, STL
{ S7_Optimized_Access := 'FALSE' }
AUTHOR : MS
// Kopieren Rezeptparameter
// stored: AutoNumber false
   VAR_INPUT
      Pos_Nr : USInt;
      WT_DB_Nr : Word;
   END_VAR
   VAR_TEMP
      WT_DB : Word;
      Par_Nr : Int;
      Schrittweite : Int;
      Par_ID : USInt;
      Cmd : USInt;
   END_VAR
BEGIN

NETWORK
TITLE = Polwender verwenden
//Positionsadresse laden
      L     #Pos_Nr;
      L     0;
      ==I;
      BEC;

//WT DB laden
      L     #WT_DB_Nr;
      T     #WT_DB;
//Pointer auf Befehl 1 setzen
      OPN   DB [#WT_DB];
      L     %DBW0;  //max. Anzahl
      L     %DBW48;  //Befehls-Nr
      <=I;
      BEC;
      L     %DBW48;  //Befehls-Nr
      L     %DBW4;  //Länge
      *I;
      L     %DBW2;  //Offset
      +I;
      SLD   3;
      LAR1;
      L     DBB [AR1, P#0.0];  //akt_Cmd
      T     #Cmd;
      L     DBW [AR1, P#6.0];  //Param-Pntr
      T     %DBW46;  //Pointer aktuell

//------------------------
//Parameter Kopieren
//------------------------
      L     0;
      T     #Par_Nr;
RET:  L     #Pos_Nr;
      L     1;
      -I;
      L     "DB_PAR_ID".Leng;
      *I;
      L     "DB_PAR_ID".Offset;
      +I;
      L     #Par_Nr;
      +I;
      SLD   3;
      LAR1;
      OPN   "DB_PAR_ID";
      L     DBB [AR1, P#0.0];
      T     #Par_ID;
//PARAMETERADRESSE LADEN
      OPN   DB [#WT_DB];
      L     %DBW46;  //Pointer aktuell
      SLD   3;
      LAR2;

      OPN   "DB_POS";
      L     #Par_ID;
      JL    list;
      JU    ende;
      JU    ID1;  //1 Expozeit
      JU    ID2;  //2 Variante
list: JU    ende;
//------------------------------
//Sollexpo
//------------------------------
ID1:  L     4;
      T     #Schrittweite;

      L     1.0;
      L     "DB_POS".POS[0].KF_Expo;
      ==R;
      OPN   DB [#WT_DB];
      L     DBD [AR2, P#0.0];
      JC    ExOk;
      DTR;
      *R;
      RND;
ExOk: T     "DB_POS".POS[0].Soll_Expozeit;
      JU    NEXT;
//------------------------------
//Variante
//------------------------------
ID2:  L     1;
      T     #Schrittweite;
      JU    NEXT;

//-----------------------------
//nächsten Parameter laden
//-----------------------------
NEXT: OPN   DB [#WT_DB];
      L     %DBW46;
      L     #Schrittweite;
      +I;
      T     %DBW46;

      L     #Par_Nr;
      L     1;
      +I;
      T     #Par_Nr;
      L     "DB_PAR_ID".Leng;
      <I;
      JC    RET;
ende: BE;

END_FUNCTION

FUNCTION "FC_Pos_Behandlung" : Void   // FC52, STL
TITLE = Positionsbehandlung
{ S7_Optimized_Access := 'FALSE' }
// Bearbeitung (Fertigmeldung/Vorruf/Räumung)
// stored: AutoNumber false
   VAR_INPUT
      Pos_Nr : USInt;
      send_DBEvt : Bool;   // Datenbank-Events senden
   END_VAR
   VAR_TEMP
      Fertigzeit : DInt;
      akt_Systime : DInt;
      Toleranz : DInt;
      Restzeit : DInt;   // Zeit bis fertig
      WT_Lang : DInt;
      WT_Nr_lang : DWord;
      StandAdr : DWord;
      Param : DWord;
      MW_Strom : Real;
      WT_DB_NR : Word;   // WT Datenbaustein-Nummer
      Standinfo : Byte;   // Beladestandinformation
      inf1 : Byte;
      Alex_ok : Bool;
      WT_nok : Bool;
   END_VAR
BEGIN

NETWORK
TITLE = Initialisierung
// allgemeine Behandlung
      A     "DB_POS".POS[0].Ziel;
      A     "DB_POS".POS[0].QT_FW_Ruf;
      R     "DB_POS".POS[0].QT_FW_Ruf;

      A     "DB_POS".POS[0].Sperre_in;
      R     "DB_POS".POS[0].Vorsperre;

      A     "DB_POS".POS[0].Ziel;
      JC    leer;
      L     "DB_POS".POS[0].WT_DB;
      T     "DB_POS".POS[0].next_WT;


NETWORK
TITLE = Position räumen
// Löschen der Position bei WT_DB==0
leer: L     "DB_POS".POS[0].WT_DB;
      L     0;
      <>I;
      JC    WTin;
//--------------------------------
//Position bereinigen
//--------------------------------
      R     "DB_POS".POS[0].WT_neu;
      R     "DB_POS".POS[0].AL_Expo;
      R     "DB_POS".POS[0].berechnet;
      R     "DB_POS".POS[0].belegt;
      R     "DB_POS".POS[0].Bearbeitung;
      R     "DB_POS".POS[0].Vorruf;
      R     "DB_POS".POS[0].fertig;
      R     "DB_POS".POS[0].Trommel;
      R     "DB_POS".POS[0].lngsm_Hub;
      R     "DB_POS".POS[0].ignor_Exp;
      R     "DB_POS".POS[0].B_Takte_Null;
      R     "DB_POS".POS[0].Opt_Abgelehnt;
      R     "DB_POS".POS[0].Belegt_KS;
      R     "DB_POS".POS[0].Belegt_LS;
      R     "DB_POS".POS[0].Belegt_GO;

      L     0;
      T     "DB_POS".POS[0].WT_Befx;
      T     "DB_POS".POS[0].WT_Nr_lang;
      T     "DB_POS".POS[0].Restzeit;
      T     "DB_POS".POS[0].Resttakte;
      T     "DB_POS".POS[0].Korr_Restzeit;
      T     "DB_POS".POS[0].WT_Stangen_Nr;
      T     "DB_POS".POS[0].WT_Typ;
      T     "DB_POS".POS[0].Korr_Restzeit;
      T     "DB_POS".POS[0].WaitTime;

      AN    #send_DBEvt;
      JC    nevt;
      T     "DB_POS".POS[0].Verweilzeit;

nevt: AN    "DB_POS".POS[0].Optipos;
      JC    Copy;
      T     "DB_POS".POS[0].Soll_Expozeit;
      JU    Copy;


NETWORK
TITLE = WT ist in der Position
//--------------------------------------
//Warenträger-DB ermitteln
//--------------------------------------
WTin: S     "DB_POS".POS[0].belegt;
      L     "DB_POS".POS[0].WT_DB;
      L     100;
      +I;
      T     #WT_DB_NR;

      L     "DB_POS".POS[0].WT_Nr_lang;
      L     0;
      <>D;
      JC    bbb;
      T     "DB_POS".POS[0].Verweilzeit;
bbb:  NOP   0;
//--------------------------------------
//Überschreitung Expotoleranz prüfen
//---------------------------------
      L     0;
      L     "DB_POS".POS[0].Prio_Pos;
      ==I;
      =     #Alex_ok;

      A     "DB_ANLAGE".config.Anl_getaktet;
      L     "DB_ANLAGE".config.Taktzeit_typ;
      JC    TTol;
      L     "DB_POS".POS[0].ExpoToleranz;
TTol: T     #Toleranz;

      L     #Toleranz;
      DTR;
      L     1.5;
      *R;
      RND;
      L     "DB_POS".POS[0].Soll_Expozeit;
      +D;
      L     "DB_POS".POS[0].WaitTime;
      +D;
      L     "DB_POS".POS[0].Verweilzeit;
      <D;
      SET;
      S     #Alex_ok;

      L     #Toleranz;
      L     30;
      <I;
      JC    korT;
      CAC;
korT: L     #Toleranz;
      L     "DB_POS".POS[0].Soll_Expozeit;
      +D;
      L     "DB_POS".POS[0].WaitTime;
      +D;
      L     "DB_POS".POS[0].Verweilzeit;
      <D;
      AN    "DB_POS".POS[0].Quelle;
      S     "DB_POS".POS[0].AL_Expo;

      L     #Toleranz;
      L     "DB_POS".POS[0].Soll_Expozeit;
      +D;
      L     "DB_POS".POS[0].WaitTime;
      +D;
      L     "DB_POS".POS[0].Verweilzeit;
      >=D;
      O(;
      L     "DB_POS".POS[0].Typ;
      L     0;
      <>I;
      );
      R     "DB_POS".POS[0].AL_Expo;

      AN    "DB_POS".POS[0].AL_Expo;
      R     "DB_POS".POS[0].MD_Alex;

      L     "DB_POS".POS[0].WT_Nr_lang;
      T     #WT_Nr_lang;

      AN    "DB_POS".POS[0].AL_Expo;
      O     "DB_POS".POS[0].MD_Alex;
      ON    "DB_POS".POS[0].yALEX;
      ON    #Alex_ok;
      JC    alok;
      S     "DB_POS".POS[0].MD_Alex;
      OPN   DB [#WT_DB_NR];
      S     %DBX22.3;  //"DB_WT1".WT_nok

alok: NOP   0;

//--------------------------------------
//Prüfung auf mitgebrachte
//Korrekturzeit am WT
//--------------------------------------
      L     0;  //Savetime löschen
      L     "DB_POS".POS[0].Typ;
      ==I;
      AN    "DB_POS".POS[0].Optipos;
      JC    SVT;
      OPN   DB [#WT_DB_NR];
      L     0;
      T     %DBD50;  //SaveTime einer Zwangsräumung
SVT:  NOP   0;

      L     "DB_POS".POS[0].Soll_Expozeit;
      L     "DB_POS".POS[0].WaitTime;
      +D;
      L     "DB_POS".POS[0].Verweilzeit;
      -D;
      T     #Restzeit;
      JPZ   rest;
      L     0;
rest: T     "DB_POS".POS[0].Restzeit;

      OPN   DB [#WT_DB_NR];
      L     %DBD50;  //SaveTime einer Zwangsräumung
      L     "DB_POS".POS[0].ExpoToleranz;
      >D;  //gesicherte Zeit zu groß --> max. um Toleranz erhöhen
      JC    KorP;
      CAC;
KorP: L     #Restzeit;
      +D;
      JPZ   nKor;
      L     0;
nKor: T     #Restzeit;
      T     "DB_POS".POS[0].Korr_Restzeit;

//--------------------------------------
//Vorruf
//--------------------------------------
      L     0;
      L     "DB_POS".POS[0].T_Vorruf;
      <I;
      O     "DB_ANLAGE".config.Anl_getaktet;
      JC    VT;
      L     "DB_Fahr-Hubzeit".UZ_typ;
      L     2.0;
      *R;
      RND;
VT:   L     #Restzeit;
      >=D;
      A(;
      AN    "DB_POS".POS[0].Optipos;
      O     "DB_POS".POS[0].berechnet;
      ON(;
      A     "DB_ANLAGE".config.EntmFromOpt;
      A     "DB_POS".POS[0].INE;  //in die Entmetallisierung
      O     "DB_POS".POS[0].INA;  //in die Anlage
      );
      O     "DB_ANLAGE".config.Anl_getaktet;
      );
      =     "DB_POS".POS[0].Vorruf;

//--------------------------------------
//Fertigmeldung
//--------------------------------------
      L     16#0000_0000;
      L     #Restzeit;
      ==D;
      A(;
      AN    "DB_POS".POS[0].Optipos;
      O     "DB_POS".POS[0].berechnet;
      ON(;
      A     "DB_ANLAGE".config.EntmFromOpt;
      A     "DB_POS".POS[0].INE;  //in die Entmetallisierung
      O     "DB_POS".POS[0].INA;  //in die Anlage
      );
      O     "DB_ANLAGE".config.Anl_getaktet;
      );
      =     "DB_POS".POS[0].fertig;

//-------------------------------
//Expozeit abgelaufen
//-------------------------------
      AN    "DB_POS".POS[0].fertig;
      ON    "DB_POS".POS[0].Bearbeitung;
      JC    RUN;
      R     "DB_POS".POS[0].Bearbeitung;



NETWORK
TITLE = Expozeit ist aktiv
//-----------------------------
//Eine gesetzte Sperre löscht
//die Zielinformation am WT
//D.h. Freigabe des Ziels
//-----------------------------
RUN:  L     "DB_POS".POS[0].Typ;
      L     10;  //Quertransport
      ==I;
      JC    reWT;

      AN    "DB_POS".POS[0].Sperre_out;
      AN    "DB_POS".POS[0].notFG_out;
      JC    reWT;

      OPN   DB [#WT_DB_NR];
      L     0;  //Löschen der Zielinfo
      T     %DBB36;  //"DB_WT1".End_Ziel_Pos
      T     %DBB37;  //"DB_WT1".End_Ziel_Reihe

//----------------------------------
//Übernahme WT-Typ u. Stangen-Nr.
//----------------------------------
reWT: OPN   DB [#WT_DB_NR];
      L     %DBB35;  //"DB_WT1".WT_Typ
      T     "DB_POS".POS[0].WT_Typ;
      OPN   DB [#WT_DB_NR];
      L     %DBB14;
      T     "DB_POS".POS[0].WT_Stangen_Nr;
      OPN   DB [#WT_DB_NR];
      L     %DBB54;  //"DB_WT1".Bereichstakte
      L     0;
      ==I;
      A(;
      L     %DBD6;  //"DB_WT1".WT_NR_lang
      L     0;
      >D;
      );
      =     "DB_POS".POS[0].B_Takte_Null;

//----------------------------------
//Check ob LeerWT in Position
//----------------------------------
      OPN   DB [#WT_DB_NR];
      L     %DBD10;  //Oberfläche
      T     "DB_POS".POS[0].KF_A;
      L     0.0;
      ==R;
      =     "DB_POS".POS[0].Leer_WT;

//----------------------------------
//Trockneranforderung rücksetzen
//----------------------------------
      L     "DB_POS".POS[0].Typ;
      L     5;  //Speicher
      ==I;
      O     "DB_POS".POS[0].Leer_WT;
      OPN   DB [#WT_DB_NR];
      R     %DBX20.1;  //"DB_WT1".UT_Anforderung

//------------------------------------
//Hilfsmerker WT am QT/FW rücksetzen
//------------------------------------
      OPN   DB [#WT_DB_NR];
      L     0;
      T     %DBB21;  //gemerkte Ziel-Position
      SET;
      R     %DBX18.6;  //am FW
      R     %DBX18.7;  //im QT

//----------------------------------
//Richtungsbits aktualisieren
//----------------------------------
      L     "DB_POS".POS[0].Typ;
      L     0;  //Anlagenbad
      <>I;
      JC    Sbit;
      OPN   DB [#WT_DB_NR];

      A     %DBX18.1;  //in die Anlage
      R     %DBX18.1;  //in die Anlage
      S     %DBX18.3;  //aus der Anlage

      A     %DBX18.2;  //in die Entmetallisierung
      R     %DBX18.2;  //in die Entmetallisierung
      S     %DBX18.4;  //aus der Entmetallisierung

//------------------------------------
//Hubinformation für FW bereit stellen
//------------------------------------
Sbit: OPN   DB [#WT_DB_NR];
      A     %DBX22.1;  //langsam Heben
      =     "DB_POS".POS[0].lngsm_Hub;

      OPN   DB [#WT_DB_NR];
      L     %DBB18;
      OPN   "DB_POS";
      T     %DBB87;  //  "DB_POS".POS[0].Speicherbits

//------------------------------------
//Automatikposition Daten sichern
//------------------------------------
      OPN   DB [#WT_DB_NR];
      L     %DBB19;
      L     %DBB15;
      <>I;
      JC    Copy;


      OPN   DB [#WT_DB_NR];
      L     %DBB54;  //"DB_WT1".Bereichstakte
      T     %DBB24;  //"DB_WT1".Alt_Bereichstakte

      A     %DBX20.4;  //"DB_WT1".TW_Pos
      =     %DBX25.0;  //"DB_WT1".Alt_TW_Pos

      L     "DB_POS".POS[0].Verweilzeit;
      OPN   DB [#WT_DB_NR];
      T     %DBD26;  //VERWEILZEIT AM WT

      L     "DB_POS".POS[0].WT_Befx;
      OPN   DB [#WT_DB_NR];
      T     %DBB23;  //Befehlsindex


NETWORK
TITLE = Kopieren der Daten für den Übersichts-DB
//------------------------------------
//Standinformationen auslesen
//------------------------------------
Copy: L     "DB_POS".POS[0].WT_Nr_lang;
      T     #WT_Lang;

      L     0;
      L     "DB_POS".POS[0].Stand_Nr;
      ==I;
      JC    NoBE;  //kein Be- Entladestand
      L     "DB_BE_Stand".Anzahl;
      >I;
      JC    NoBE;
      CAC;
      DEC   1;
      L     "DB_BE_Stand".leng;
      *D;
      L     "DB_BE_Stand".Offset;
      +D;
      L     1;
      +D;
      SLD   3;
      T     #StandAdr;

      OPN   "DB_BE_Stand";
      L     DBB [#StandAdr];
      T     #Standinfo;

      L     0;
      L     #WT_Lang;
      <>D;
      JC    nalt;
      L     #StandAdr;
      SRD   3;
      +     5;
      SLD   3;
      T     #StandAdr;

      OPN   "DB_BE_Stand";
      L     DBD [#StandAdr];
      T     #WT_Lang;

nalt: L     "DB_POS".POS[0].WT_Nr_lang;
      L     0;
      ==D;
      JC    wtr;
      L     #Standinfo;
      L     16#04;
      OW;
      T     #Standinfo;
      JU    wtr;

NoBE: L     0;
      T     #Standinfo;

//------------------------------------
//Daten für Übersichts-DB
//------------------------------------
wtr:  SET;
      R     #WT_nok;

      L     "DB_Panel_OVERVIEW".Systime;
      T     #akt_Systime;
      L     0;
      T     #Fertigzeit;

      L     #Pos_Nr;
      L     1;
      -I;
      L     "DB_Panel_OVERVIEW".Leng;
      *I;
      L     "DB_Panel_OVERVIEW".Offset;
      +I;
      SLD   3;
      LAR1;
      L     "DB_POS".POS[0].WT_Nr_lang;
      L     #WT_Lang;
      OPNDI "DB_Panel_OVERVIEW";  //"DB_PC_OVERVIEW"
      T     DID [AR1, P#0.0];
      L     0;
      L     "DB_POS".POS[0].WT_DB;
      T     DIB [AR1, P#4.0];
      ==I;
      JC    wtr1;
      +     100;
      T     #WT_DB_NR;
      OPN   DB [#WT_DB_NR];
      L     %DBD30;  //"DB_WT1".Fertigzeitpunkt
      T     #Fertigzeit;
      A     %DBX22.3;  //"DB_WT1".WT_nok
      =     #WT_nok;

      L     %DBB63;  //"DB_WT1".WT_Kenn
wtr1: T     DIB [AR1, P#15.0];  //Sonderfkt

      L     "DB_POS".POS[0].WT_Stangen_Nr;
      T     DIB [AR1, P#5.0];
      L     "DB_POS".POS[0].WT_Typ;
      T     DIB [AR1, P#21.0];
      L     "DB_POS".POS[0].Soll_Expozeit;
      T     DID [AR1, P#6.0];

// Rücklaufende Expozeiten
      L     "DB_POS".POS[0].Soll_Expozeit;
      L     "DB_POS".POS[0].Verweilzeit;
      -D;
      T     DID [AR1, P#10.0];

      L     #Standinfo;
      T     DIB [AR1, P#14.0];
      OPN   "DB_POS";
      L     %DBB87;  //  "DB_POS".POS[0].Speicherbits
      T     DIB [AR1, P#16.0];
      A     "DB_POS".POS[0].Warnung;
      =     DIX [AR1, P#16.6];
      A     "DB_POS".POS[0].Alarm;
      =     DIX [AR1, P#16.7];
      A     "DB_POS".POS[0].belegt;
      =     DIX [AR1, P#17.0];
      A     "DB_POS".POS[0].Trommel;
      =     DIX [AR1, P#17.1];
      A     "DB_POS".POS[0].Leer_WT;
      =     DIX [AR1, P#17.2];
      A     "DB_POS".POS[0].Vorruf;
      =     DIX [AR1, P#17.3];
      A     "DB_POS".POS[0].fertig;
      =     DIX [AR1, P#17.4];
      A     "DB_POS".POS[0].Sperre_in;
      =     DIX [AR1, P#17.5];
      A     "DB_POS".POS[0].Sperre_FW;
      =     DIX [AR1, P#17.6];
      A     "DB_POS".POS[0].Sperre_out;
      =     DIX [AR1, P#17.7];
      L     "DB_POS".POS[0].WT_Befx;
      T     DIW [AR1, P#18.0];
      A     "DB_POS".POS[0].Vorsperre;
      =     DIX [AR1, P#20.0];
      A     "DB_POS".POS[0].Spr_Off;  //Dummy in Dummyposition
      =     DIX [AR1, P#20.1];
      A     "DB_POS".POS[0].Opt_Abgelehnt;
      =     DIX [AR1, P#20.2];
      A     "DB_POS".POS[0].Dkl_auf_Pos;
      =     DIX [AR1, P#20.3];  //Deckel auf Pos.
      A     "DB_POS".POS[0].AL_Expo;
      A     "DB_POS".POS[0].yALEX;
      =     DIX [AR1, P#20.4];
      A     "DB_POS".POS[0].Expo_Off;
      =     DIX [AR1, P#20.5];
      L     "DB_POS".POS[0].Verweilzeit;
      T     DID [AR1, P#22.0];
      L     #Fertigzeit;
      T     DID [AR1, P#30.0];
      A     "DB_POS".POS[0].PendHub;
      =     DIX [AR1, P#39.4];

//------------------------------------
//Daten für Detailinformations-DB
//------------------------------------
      L     #Pos_Nr;
      L     1;
      -I;
      L     "DB_Panel_Posinfo".Leng;
      *I;
      L     "DB_Panel_Posinfo".Offset;
      +I;
      SLD   3;
      LAR1;
      L     "DB_POS".POS[0].Prio_Pos;
      OPNDI "DB_Panel_Posinfo";  //"DB_PC_Posinfo"
      T     DIB [AR1, P#0.0];
      A     "DB_POS".POS[0].lngsm_IN;
      =     DIX [AR1, P#1.0];
      A     "DB_POS".POS[0].lngsm_OUT;
      =     DIX [AR1, P#1.1];
      A     "DB_POS".POS[0].KS_erlaubt;
      =     DIX [AR1, P#20.5];
      L     "DB_POS".POS[0].Verweilzeit;
      T     DID [AR1, P#2.0];
      L     "DB_POS".POS[0].KF_A;
      T     DID [AR1, P#6.0];
      L     "DB_POS".POS[0].KF_Expo;
      T     DID [AR1, P#10.0];
      L     "DB_POS".POS[0].T_Vorruf;
      T     DIW [AR1, P#14.0];
      L     "DB_POS".POS[0].T_Pend;
      T     DIW [AR1, P#16.0];
      L     "DB_POS".POS[0].T_ATZ;
      T     DIW [AR1, P#18.0];
      L     "DB_POS".POS[0].ExpoToleranz;
      T     DID [AR1, P#56.0];

END_FUNCTION

FUNCTION "FC_WORK_TO_POS" : Void   // FC54, STL
TITLE = Arbeitsdaten zurückschreiben
{ S7_Optimized_Access := 'FALSE' }
AUTHOR : MS
// Überträgt die Positionsdaten nach der Bearbeitung wieder in den Positions-DB
// stored: AutoNumber false
   VAR_INPUT
      Akt_Pos : USInt;   // Position die geladen wird
   END_VAR
BEGIN

NETWORK
TITLE = Move Dat
// von Feld[0] -- > [akt_pos]
      CALL  MOVE
      ( IN  := "DB_POS".POS[0],
        OUT := "DB_POS".POS[#Akt_Pos]
      );

END_FUNCTION

FUNCTION "FC_WT_from_Pos" : Void   // FC57, STL
TITLE = Umladen eines Wt aus einer Pos an FW/QT
{ S7_Optimized_Access := 'FALSE' }
// Aufruf aus FW bzw. QT
// stored: AutoNumber false
   VAR_INPUT
      Pos_Nr : USInt;
      send_DBEvt : Bool;   // Datenbank-Events senden
   END_VAR
   VAR_OUTPUT
      load_ok : Bool;
   END_VAR
   VAR_IN_OUT
      WT_Nr : Byte;
      WT_Nr_lang : DWord;
   END_VAR
   VAR_TEMP
      not_load : Bool;
      WT_DB : Word;
      Param : DWord;
      MW_Strom : Real;
      MD_Nr : USInt;
      inf_1 : Byte;
   END_VAR
BEGIN

NETWORK
TITLE = 
//----------------------------
//laden der Pos und prüfen
//----------------------------
      SET;
      R     #load_ok;

      CALL  "FC_POS_TO_WORK"
      ( Akt_Pos  := #Pos_Nr,
        not_load := #not_load
      );

      A     #not_load;
      BEC;

      L     0;
      L     "DB_POS".POS[0].WT_DB;
      >=I;
      BEC;

//----------------------------
//Umladen erlaubt
//----------------------------
      S     #load_ok;
      T     #WT_Nr;
      L     100;
      +I;
      T     #WT_DB;

      L     "DB_POS".POS[0].WT_Nr_lang;
      T     #WT_Nr_lang;

//----------------------------
//Abbruch --> Restzeit sichern
//----------------------------
      AN    "DB_POS".POS[0].ignor_Exp;
      L     0;
      JC    noZw;
      L     "DB_POS".POS[0].Restzeit;
noZw: OPN   DB [#WT_DB];
      L     %DBD50;  //Sicherung der fehlenden Expozeit am WT
      +D;
      T     %DBD50;  //Sicherung der fehlenden Expozeit am WT

      AN    #send_DBEvt;
      JC    noDB;

//----------------------------
//WT in Pos löschen
//----------------------------
noDB: L     0;
      T     "DB_POS".POS[0].WT_DB;  //WT_Nr_Kurz im Bad
      T     "DB_POS".POS[0].WT_Nr_lang;  //WT_Nr lang im Bad

//----------------------------
//Position aktualisieren
//----------------------------
      CALL  "FC_Pos_Behandlung"
      ( Pos_Nr     := #Pos_Nr,
        send_DBEvt := #send_DBEvt
      );
//-------------------------------
//zurückladen der PosDaten
//-------------------------------
      CALL  "FC_WORK_TO_POS"
      ( Akt_Pos := #Pos_Nr
      );

END_FUNCTION

FUNCTION "FC_Beladen" : Void   // FC43, STL
TITLE = Be-/Entladestand
{ S7_Optimized_Access := 'FALSE' }
// Datenbasis für Beladestandhandling DB4
// stored: AutoNumber false
   VAR_INPUT
      Stand_Nr : Int;   // Nummer des Beladestandes
      E_Belegt : Bool;   // WT erkannt (bei nicht vorhanden auf TRUE setzen)
      E_S_innen : Bool;   // Wagen innerer Sensor ok (bei nicht vorhanden auf TRUE setzen)
      E_S_aussen : Bool;   // Wagen äußerer Sensor ok (bei nicht vorhanden auf TRUE setzen)
      E_S_verriegelt : Bool;   // Standbedienung erlaubt (bei nicht vorhanden auf TRUE setzen)
      E_Freigabe : Bool;   // Freigabetaster aus Stand-DB (bei nicht vorhanden auf TRUE setzen)
      Auto_Delete : Bool;   // automatisches löschen fertiger WT
      ext_Delete : Bool;   // löschen durch externe Anforderung
      Del_All : Bool;   // 0=Programm löschen 1=gesamten WT löschen
      Afg_WT_Nr : Bool;   // Aufgabe auch bei WT_Nr_lang<>0 erlaubt
      Del_count : Int;   // Zeit nach der Wt gelöscht wird in s
   END_VAR
   VAR_TEMP
      WT_DB : Int;
      Pos_Nr : USInt;
      WT_Nr : Byte;
      WT_Nr_lang : DWord;
      "Return" : Bool;
      kein_Korb : Bool;
   END_VAR
BEGIN

NETWORK
TITLE = Initialisierung
// Berechnung der Arbeitsbereiche
// und initialisieren temporärer Variablen
//---------------------------------
//Zeiger auf Stand (DB4) berechnen
//---------------------------------
      L     0;
      L     #Stand_Nr;
      ==I;
      BEC;
      L     "DB_BE_Stand".Anzahl;
      >I;
      BEC;

      A     #Del_All;
      =     "DB_BE_Stand".Stand[#Stand_Nr].Del_All;
      A     #Auto_Delete;
      =     "DB_BE_Stand".Stand[#Stand_Nr].Auto_Delete;
      A     #Afg_WT_Nr;
      =     "DB_BE_Stand".Stand[#Stand_Nr].Afg_WT_Nr;

      L     "DB_BE_Stand".Stand[#Stand_Nr].Pos_Nr;
      T     #Pos_Nr;


NETWORK
TITLE = Bearbeitung Sperren und Freigaben
//----------------------------
//Signal FW kommt
//----------------------------
      A     "DB_POS".POS[#Pos_Nr].FW_kommt;
      =     "DB_BE_Stand".Stand[#Stand_Nr].OUT_FW_kommt;

//----------------------------
//Stand ist leer
//----------------------------
      L     "DB_POS".POS[#Pos_Nr].WT_DB;
      L     0;
      ==I;
      AN    #Del_All;
      O(;
      AN    #E_Belegt;
      A     #Del_All;
      );
      =     "DB_BE_Stand".Stand[#Stand_Nr].kein_WT;

//----------------------------
//WT bereits aufgegeben
//----------------------------
      L     0;
      L     "DB_POS".POS[#Pos_Nr].WT_DB;
      ==I;
      JC    goon;
      +     100;
      T     #WT_DB;
      OPN   DB [#WT_DB];
      AN(;
      L     %DBW48;  //"DB_WTx".B_PNTER
      L     1;
      >I;
      );
goon: A(;
      L     "DB_POS".POS[#Pos_Nr].WT_Nr_lang;
      L     0;
      <>D;
      );
      A     "DB_POS".POS[#Pos_Nr].belegt;
      A     "DB_POS".POS[#Pos_Nr].INA;
      =     "DB_BE_Stand".Stand[#Stand_Nr].WT_aufgegeben;

//----------------------------
//Aufgabe erlauben
//----------------------------
      L     "DB_POS".POS[#Pos_Nr].WT_Nr_lang;
      L     0;
      ==D;
      O     #Afg_WT_Nr;
      A     #E_S_aussen;
      AN    "DB_POS".POS[#Pos_Nr].FW_Hebt;
      AN    "DB_POS".POS[#Pos_Nr].FW_Senkt;
      AN    "DB_BE_Stand".Stand[#Stand_Nr].kein_WT;
      =     "DB_BE_Stand".Stand[#Stand_Nr].Aufgabe_erlaubt;

//----------------------------
//Sperre FW
//----------------------------
      A     #E_S_innen;
      X     #E_S_aussen;
      NOT;
      =     "DB_BE_Stand".Stand[#Stand_Nr].OUT_Sperre_FW;
//----------------------------
//Einfahrsperre
//----------------------------
      L     "DB_POS".POS[#Pos_Nr].WT_DB;
      L     0;
      <>I;
      O(;
      A     #E_Belegt;
      A     #Del_All;
      );
      ON    #E_S_innen;
      O     #E_S_aussen;
      ON    #E_S_verriegelt;
      =     "DB_BE_Stand".Stand[#Stand_Nr].OUT_Sperre_in;

//----------------------------
//Ausfahrsperre
//----------------------------
      L     "DB_POS".POS[#Pos_Nr].WT_DB;
      L     0;
      ==I;
      O(;
      AN    #E_Belegt;
      A     #Del_All;
      );
      ON    #E_S_innen;
      O     #E_S_aussen;
      ON    #E_S_verriegelt;
      ON    "DB_BE_Stand".Stand[#Stand_Nr].WT_aufgegeben;
      =     "DB_BE_Stand".Stand[#Stand_Nr].OUT_Sperre_out;


NETWORK
TITLE = Löschen eines WT
// WTs werden gelöscht, wenn der Wagen abgezogen wird
// oder ein fertiger WT abgelegt wird.
// Ein WT wird nicht gelöscht, während der FW hebt/senkt oder der Belegtsensor
// ausfällt.
      L     "DB_POS".POS[#Pos_Nr].WT_DB;
      L     0;
      <>I;
      JC    wtok;
      T     "DB_BE_Stand".Stand[#Stand_Nr].last_WT;
wtok: NOP   0;
//----------------------------
//Stand wird gerade bedient
//----------------------------
      A     "DB_POS".POS[#Pos_Nr].FW_Hebt;
      O     "DB_POS".POS[#Pos_Nr].FW_Senkt;
      BEC;

//----------------------------
//Korb wird entfernt
//----------------------------
      A     #E_S_aussen;
      AN    #E_Belegt;
      =     #kein_Korb;
      JC    Del;
//----------------------------
//manuelles Löschen (Zeit)
//----------------------------
      A     #ext_Delete;
      JC    Del;
//----------------------------
//Automatisches Löschen (Zeit)
//----------------------------
      AN    #Auto_Delete;
      BEC;
      A     "DB_POS".POS[#Pos_Nr].OUTA;
      JC    Wait;

      L     "DB_POS".POS[#Pos_Nr].WT_Befx;
      L     0;
      <>I;
      JC    Wait;
      L     #Del_count;  //Wartezeit laden
      T     "DB_BE_Stand".Stand[#Stand_Nr].Del_Count;
      BE;

Wait: L     "DB_BE_Stand".Stand[#Stand_Nr].Del_Count;
      L     0;
      <=I;
      JC    Del;  //Zeit abgelaufen
      AN    "Imp_1Hz";  //Sekundentakt
      BEC;
      CAC;
      DEC   1;
      T     "DB_BE_Stand".Stand[#Stand_Nr].Del_Count;
      BE;

//----------------------------
//Löschvorgang
//----------------------------
Del:  L     "DB_POS".POS[#Pos_Nr].WT_DB;
      L     0;
      ==I;
      O(;
      L     "DB_POS".POS[#Pos_Nr].WT_Nr_lang;
      L     0;
      ==D;
      AN    #Del_All;
      );
      BEC;  //bereits gelöscht

      CALL  "FC_WT_from_Pos"
      ( Pos_Nr     := #Pos_Nr,
        send_DBEvt := FALSE,
        load_ok    := #"Return",
        WT_Nr      := #WT_Nr,
        WT_Nr_lang := #WT_Nr_lang
      );  //Position bereinigen

      AN    #"Return";  //Ladevorgang mißlungen
      BEC;

